SPLINE
SPL {X  -145.877, Y  +737.201, Z    +0.000, E1   -34.468, E3 +267717.611}
SPL {X  -152.550, Y  +719.721, Z    +0.000, E1   -27.728, E3 +267733.100}
SPL {X  -157.145, Y  +701.536, Z    +0.000, E1   -19.368, E3 +267742.554}
SPL {X  -159.035, Y  +688.952, Z    +0.000, E1   -12.676, E3 +267746.596}
SPL {X  -159.756, Y  +680.154, Z    +0.000, E1    -7.520, E3 +267748.322}
SPL {X  -159.986, Y  +672.560, Z    +0.000, E1    -2.636, E3 +267749.220}
SPL {X  -159.990, Y  +668.344, Z    +0.000, E1    +0.618, E3 +267749.486}
SPL {X  -159.990, Y  +664.070, Z    +0.000, E1    +5.025, E3 +267749.815}
SPL {X  -159.990, Y  +656.953, Z    +0.000, E1   +13.960, E3 +267750.881}
SPL {X  -159.990, Y  +644.589, Z    +0.000, E1   +29.011, E3 +267754.293}
SPL {X  -159.990, Y  +605.095, Z    +0.000, E1   +49.514, E3 +267779.383}
SPL {X  -159.990, Y  +543.998, Z    +0.000, E1   +54.483, E3 +267845.373}
SPL {X  -159.990, Y  +535.878, Z    +0.000, E1   +54.465, E3 +267857.708}
SPL {X  -159.990, Y  +529.394, Z    +0.000, E1   +54.464, E3 +267867.538}
SPL {X  -159.990, Y  +521.536, Z    +0.000, E1   +54.480, E3 +267879.419}
SPL {X  -159.990, Y  +514.089, Z    +0.000, E1   +54.461, E3 +267890.732}
SPL {X  -159.990, Y  +506.373, Z    +0.000, E1   +54.484, E3 +267902.368}
SPL {X  -159.990, Y  +497.571, Z    +0.000, E1   +54.478, E3 +267915.711}
SPL {X  -159.990, Y  +490.343, Z    +0.000, E1   +54.468, E3 +267926.676}
SPL {X  -159.990, Y  +483.191, Z    +0.000, E1   +54.478, E3 +267937.492}
SPL {X  -159.990, Y  +471.543, Z    +0.000, E1   +55.096, E3 +267951.120}
SPL {X  -159.990, Y  +443.253, Z    +0.000, E1   +59.297, E3 +267962.552}
SPL {X  -159.990, Y  +438.044, Z    +0.000, E1   +58.687, E3 +267973.407}
SPL {X  -159.990, Y  +431.936, Z    +0.000, E1   +57.955, E3 +267986.227}
SPL {X  -159.990, Y  +427.860, Z    +0.000, E1   +57.091, E3 +267997.291}
SPL {X  -159.990, Y  +424.653, Z    +0.000, E1   +55.901, E3 +268009.596}
SPL {X  -159.990, Y  +418.232, Z    +0.000, E1   +55.048, E3 +268024.389}
SPL {X  -159.990, Y  +410.722, Z    +0.000, E1   +54.900, E3 +268036.372}
SPL {X  -159.990, Y  +402.790, Z    +0.000, E1   +54.930, E3 +268048.147}
SPL {X  -159.990, Y  +391.119, Z    +0.000, E1   +54.948, E3 +268065.524}
SPL {X  -159.951, Y  +378.972, Z    +0.000, E1   +54.929, E3 +268083.703}
SPL {X  -159.499, Y  +369.977, Z    +0.000, E1   +54.827, E3 +268097.615}
SPL {X  -158.803, Y  +363.045, Z    +0.000, E1   +54.709, E3 +268108.684}
SPL {X  -157.966, Y  +357.131, Z    +0.000, E1   +54.559, E3 +268118.386}
SPL {X  -156.775, Y  +350.586, Z    +0.000, E1   +54.373, E3 +268129.360}
SPL {X  -155.027, Y  +342.959, Z    +0.000, E1   +54.074, E3 +268142.533}
SPL {X  -152.882, Y  +335.340, Z    +0.000, E1   +53.695, E3 +268156.076}
SPL {X  -151.019, Y  +329.680, Z    +0.000, E1   +53.334, E3 +268166.433}
SPL {X  -149.351, Y  +325.131, Z    +0.000, E1   +53.025, E3 +268174.877}
SPL {X  -147.860, Y  +321.391, Z    +0.000, E1   +52.740, E3 +268181.930}
SPL {X  -145.914, Y  +316.881, Z    +0.000, E1   +52.402, E3 +268190.499}
SPL {X  -142.795, Y  +310.344, Z    +0.000, E1   +51.829, E3 +268203.155}
SPL {X  -132.354, Y  +292.616, Z    +0.000, E1   +44.164, E3 +268301.567}
ENDSPLINE

SPLINE
SPL {X  -150.910, Y  +329.369, Z    +0.000, E1   +29.678, E3 +268373.963}
SPL {X  -156.396, Y  +348.778, Z    +0.000, E1   +21.134, E3 +268385.606}
SPL {X  -158.554, Y  +361.116, Z    +0.000, E1   +14.883, E3 +268390.060}
SPL {X  -159.881, Y  +376.607, Z    +0.000, E1    +5.865, E3 +268393.469}
SPL {X  -159.990, Y  +383.659, Z    +0.000, E1    +1.050, E3 +268394.150}
SPL {X  -159.990, Y  +387.327, Z    +0.000, E1    -2.137, E3 +268394.383}
SPL {X  -159.990, Y  +390.622, Z    +0.000, E1    -5.876, E3 +268394.676}
SPL {X  -159.990, Y  +394.493, Z    +0.000, E1   -10.512, E3 +268395.199}
SPL {X  -159.990, Y  +401.377, Z    +0.000, E1   -19.398, E3 +268396.653}
SPL {X  -159.990, Y  +411.365, Z    +0.000, E1   -30.630, E3 +268399.862}
SPL {X  -159.990, Y  +450.467, Z    +0.000, E1   -50.183, E3 +268423.511}
SPL {X  -159.990, Y  +509.934, Z    +0.000, E1   -54.923, E3 +268486.130}
SPL {X  -159.990, Y  +516.848, Z    +0.000, E1   -54.930, E3 +268496.418}
SPL {X  -159.990, Y  +524.818, Z    +0.000, E1   -54.933, E3 +268508.290}
SPL {X  -159.990, Y  +532.100, Z    +0.000, E1   -54.924, E3 +268519.143}
SPL {X  -159.990, Y  +539.391, Z    +0.000, E1   -54.933, E3 +268529.995}
SPL {X  -159.990, Y  +546.283, Z    +0.000, E1   -54.924, E3 +268540.266}
SPL {X  -159.990, Y  +553.734, Z    +0.000, E1   -54.938, E3 +268551.353}
SPL {X  -159.990, Y  +564.956, Z    +0.000, E1   -54.973, E3 +268568.024}
SPL {X  -159.990, Y  +577.902, Z    +0.000, E1   -54.969, E3 +268587.314}
SPL {X  -159.990, Y  +588.063, Z    +0.000, E1   -54.931, E3 +268602.505}
SPL {X  -159.990, Y  +595.273, Z    +0.000, E1   -54.928, E3 +268613.228}
SPL {X  -159.990, Y  +602.326, Z    +0.000, E1   -54.932, E3 +268623.729}
SPL {X  -159.990, Y  +610.296, Z    +0.000, E1   -54.937, E3 +268635.598}
SPL {X  -159.990, Y  +618.534, Z    +0.000, E1   -54.942, E3 +268647.835}
SPL {X  -159.990, Y  +628.178, Z    +0.000, E1   -54.959, E3 +268662.166}
SPL {X  -159.990, Y  +638.304, Z    +0.000, E1   -54.952, E3 +268677.255}
SPL {X  -159.990, Y  +648.272, Z    +0.000, E1   -54.961, E3 +268692.064}
SPL {X  -159.990, Y  +655.990, Z    +0.000, E1   -54.930, E3 +268703.612}
SPL {X  -159.990, Y  +665.734, Z    +0.000, E1   -54.984, E3 +268718.063}
SPL {X  -159.827, Y  +678.718, Z    +0.000, E1   -54.950, E3 +268737.591}
SPL {X  -159.222, Y  +687.156, Z    +0.000, E1   -54.792, E3 +268750.902}
SPL {X  -158.388, Y  +694.082, Z    +0.000, E1   -54.679, E3 +268762.040}
SPL {X  -157.277, Y  +700.838, Z    +0.000, E1   -54.465, E3 +268773.297}
SPL {X  -156.153, Y  +706.327, Z    +0.000, E1   -54.274, E3 +268782.633}
SPL {X  -154.917, Y  +711.470, Z    +0.000, E1   -54.052, E3 +268791.584}
SPL {X  -153.204, Y  +717.603, Z    +0.000, E1   -53.775, E3 +268802.430}
SPL {X  -151.355, Y  +723.351, Z    +0.000, E1   -53.415, E3 +268812.901}
SPL {X  -149.371, Y  +728.816, Z    +0.000, E1   -53.074, E3 +268822.992}
SPL {X  -147.376, Y  +733.767, Z    +0.000, E1   -52.671, E3 +268832.394}
SPL {X  -145.158, Y  +738.775, Z    +0.000, E1   -52.288, E3 +268841.945}
SPL {X  -142.385, Y  +744.461, Z    +0.000, E1   -51.729, E3 +268853.057}
SPL {X  -132.301, Y  +761.463, Z    +0.000, E1   -45.510, E3 +268930.796}
ENDSPLINE

SPLINE
SPL {X  -145.877, Y  +737.201, Z    +0.000, E1   -34.468, E3 +269013.907}
SPL {X  -152.550, Y  +719.721, Z    +0.000, E1   -27.728, E3 +269029.396}
SPL {X  -157.145, Y  +701.536, Z    +0.000, E1   -19.368, E3 +269038.851}
SPL {X  -159.035, Y  +688.952, Z    +0.000, E1   -12.676, E3 +269042.892}
SPL {X  -159.756, Y  +680.154, Z    +0.000, E1    -7.520, E3 +269044.618}
SPL {X  -159.986, Y  +672.560, Z    +0.000, E1    -2.636, E3 +269045.516}
SPL {X  -159.990, Y  +668.344, Z    +0.000, E1    +0.618, E3 +269045.782}
SPL {X  -159.990, Y  +664.070, Z    +0.000, E1    +5.025, E3 +269046.111}
SPL {X  -159.990, Y  +656.953, Z    +0.000, E1   +13.960, E3 +269047.177}
SPL {X  -159.990, Y  +644.589, Z    +0.000, E1   +29.011, E3 +269050.589}
SPL {X  -159.990, Y  +605.095, Z    +0.000, E1   +49.514, E3 +269075.680}
SPL {X  -159.990, Y  +546.155, Z    +0.000, E1   +54.461, E3 +269138.438}
SPL {X  -159.990, Y  +537.700, Z    +0.000, E1   +54.492, E3 +269151.202}
SPL {X  -159.990, Y  +529.394, Z    +0.000, E1   +54.464, E3 +269163.834}
SPL {X  -159.990, Y  +521.536, Z    +0.000, E1   +54.480, E3 +269175.715}
SPL {X  -159.990, Y  +514.089, Z    +0.000, E1   +54.461, E3 +269187.028}
SPL {X  -159.990, Y  +506.373, Z    +0.000, E1   +54.484, E3 +269198.664}
SPL {X  -159.990, Y  +497.571, Z    +0.000, E1   +54.478, E3 +269212.007}
SPL {X  -159.990, Y  +490.343, Z    +0.000, E1   +54.468, E3 +269222.972}
SPL {X  -159.990, Y  +483.191, Z    +0.000, E1   +54.478, E3 +269233.789}
SPL {X  -159.990, Y  +475.502, Z    +0.000, E1   +54.476, E3 +269245.438}
SPL {X  -159.990, Y  +448.520, Z    +0.000, E1   +58.543, E3 +269257.067}
SPL {X  -159.990, Y  +438.044, Z    +0.000, E1   +58.687, E3 +269269.704}
SPL {X  -159.990, Y  +431.936, Z    +0.000, E1   +57.955, E3 +269282.523}
SPL {X  -159.990, Y  +427.860, Z    +0.000, E1   +57.091, E3 +269293.587}
SPL {X  -159.990, Y  +424.653, Z    +0.000, E1   +55.901, E3 +269305.892}
SPL {X  -159.990, Y  +418.232, Z    +0.000, E1   +55.048, E3 +269320.685}
SPL {X  -159.990, Y  +410.722, Z    +0.000, E1   +54.900, E3 +269332.668}
SPL {X  -159.990, Y  +402.790, Z    +0.000, E1   +54.930, E3 +269344.443}
SPL {X  -159.990, Y  +392.953, Z    +0.000, E1   +54.918, E3 +269359.137}
SPL {X  -159.990, Y  +383.354, Z    +0.000, E1   +54.920, E3 +269373.447}
SPL {X  -159.860, Y  +376.053, Z    +0.000, E1   +54.872, E3 +269384.507}
SPL {X  -159.499, Y  +369.977, Z    +0.000, E1   +54.827, E3 +269393.911}
SPL {X  -158.803, Y  +363.045, Z    +0.000, E1   +54.709, E3 +269404.980}
SPL {X  -157.732, Y  +355.717, Z    +0.000, E1   +54.540, E3 +269417.002}
SPL {X  -156.235, Y  +348.039, Z    +0.000, E1   +54.281, E3 +269430.014}
SPL {X  -154.716, Y  +341.761, Z    +0.000, E1   +53.995, E3 +269440.971}
SPL {X  -152.882, Y  +335.340, Z    +0.000, E1   +53.695, E3 +269452.372}
SPL {X  -151.019, Y  +329.680, Z    +0.000, E1   +53.334, E3 +269462.729}
SPL {X  -149.351, Y  +325.131, Z    +0.000, E1   +53.025, E3 +269471.173}
SPL {X  -147.860, Y  +321.391, Z    +0.000, E1   +52.740, E3 +269478.226}
SPL {X  -145.914, Y  +316.881, Z    +0.000, E1   +52.402, E3 +269486.796}
SPL {X  -142.795, Y  +310.344, Z    +0.000, E1   +51.829, E3 +269499.451}
SPL {X  -132.354, Y  +292.616, Z    +0.000, E1   +44.164, E3 +269597.864}
ENDSPLINE

SPLINE
SPL {X  -150.910, Y  +329.369, Z    +0.000, E1   +29.678, E3 +269670.259}
SPL {X  -156.829, Y  +350.854, Z    +0.000, E1   +20.141, E3 +269682.812}
SPL {X  -159.049, Y  +365.169, Z    +0.000, E1   +12.580, E3 +269687.556}
SPL {X  -159.776, Y  +374.231, Z    +0.000, E1    +7.281, E3 +269689.442}
SPL {X  -159.986, Y  +381.380, Z    +0.000, E1    +2.685, E3 +269690.288}
SPL {X  -159.990, Y  +384.493, Z    +0.000, E1    +0.324, E3 +269690.496}
SPL {X  -159.990, Y  +387.327, Z    +0.000, E1    -2.137, E3 +269690.679}
SPL {X  -159.990, Y  +392.053, Z    +0.000, E1    -7.477, E3 +269691.144}
SPL {X  -159.990, Y  +396.158, Z    +0.000, E1   -12.775, E3 +269691.769}
SPL {X  -159.990, Y  +401.377, Z    +0.000, E1   -19.398, E3 +269692.950}
SPL {X  -159.990, Y  +411.365, Z    +0.000, E1   -30.630, E3 +269696.158}
SPL {X  -159.990, Y  +450.467, Z    +0.000, E1   -50.183, E3 +269719.807}
SPL {X  -159.990, Y  +509.934, Z    +0.000, E1   -54.923, E3 +269782.426}
SPL {X  -159.990, Y  +516.848, Z    +0.000, E1   -54.930, E3 +269792.714}
SPL {X  -159.990, Y  +524.818, Z    +0.000, E1   -54.933, E3 +269804.586}
SPL {X  -159.990, Y  +532.100, Z    +0.000, E1   -54.924, E3 +269815.439}
SPL {X  -159.990, Y  +539.391, Z    +0.000, E1   -54.933, E3 +269826.291}
SPL {X  -159.990, Y  +546.283, Z    +0.000, E1   -54.924, E3 +269836.562}
SPL {X  -159.990, Y  +553.734, Z    +0.000, E1   -54.938, E3 +269847.649}
SPL {X  -159.990, Y  +560.983, Z    +0.000, E1   -54.918, E3 +269858.487}
SPL {X  -159.990, Y  +567.462, Z    +0.000, E1   -54.929, E3 +269868.122}
SPL {X  -159.990, Y  +575.140, Z    +0.000, E1   -54.928, E3 +269879.554}
SPL {X  -159.990, Y  +581.046, Z    +0.000, E1   -54.920, E3 +269888.366}
SPL {X  -159.990, Y  +588.063, Z    +0.000, E1   -54.931, E3 +269898.801}
SPL {X  -159.990, Y  +595.273, Z    +0.000, E1   -54.928, E3 +269909.525}
SPL {X  -159.990, Y  +602.326, Z    +0.000, E1   -54.932, E3 +269920.025}
SPL {X  -159.990, Y  +610.296, Z    +0.000, E1   -54.937, E3 +269931.894}
SPL {X  -159.990, Y  +618.534, Z    +0.000, E1   -54.942, E3 +269944.131}
SPL {X  -159.990, Y  +625.928, Z    +0.000, E1   -54.931, E3 +269955.157}
SPL {X  -159.990, Y  +633.423, Z    +0.000, E1   -54.943, E3 +269966.299}
SPL {X  -159.990, Y  +643.352, Z    +0.000, E1   -54.966, E3 +269981.034}
SPL {X  -159.990, Y  +650.756, Z    +0.000, E1   -54.931, E3 +269992.101}
SPL {X  -159.990, Y  +658.525, Z    +0.000, E1   -54.959, E3 +270003.637}
SPL {X  -159.990, Y  +667.903, Z    +0.000, E1   -54.941, E3 +270017.668}
SPL {X  -159.953, Y  +674.920, Z    +0.000, E1   -54.918, E3 +270028.171}
SPL {X  -159.714, Y  +680.893, Z    +0.000, E1   -54.890, E3 +270037.311}
SPL {X  -159.222, Y  +687.156, Z    +0.000, E1   -54.792, E3 +270047.198}
SPL {X  -158.388, Y  +694.082, Z    +0.000, E1   -54.679, E3 +270058.336}
SPL {X  -157.277, Y  +700.838, Z    +0.000, E1   -54.465, E3 +270069.593}
SPL {X  -156.153, Y  +706.327, Z    +0.000, E1   -54.274, E3 +270078.929}
SPL {X  -154.917, Y  +711.470, Z    +0.000, E1   -54.052, E3 +270087.880}
SPL {X  -153.204, Y  +717.603, Z    +0.000, E1   -53.775, E3 +270098.726}
SPL {X  -151.355, Y  +723.351, Z    +0.000, E1   -53.415, E3 +270109.198}
SPL {X  -149.371, Y  +728.816, Z    +0.000, E1   -53.074, E3 +270119.288}
SPL {X  -146.631, Y  +735.501, Z    +0.000, E1   -52.568, E3 +270131.949}
SPL {X  -144.428, Y  +740.329, Z    +0.000, E1   -52.109, E3 +270141.303}
SPL {X  -142.385, Y  +744.461, Z    +0.000, E1   -51.729, E3 +270149.354}
SPL {X  -132.301, Y  +761.463, Z    +0.000, E1   -45.510, E3 +270227.092}
ENDSPLINE

SPLINE
SPL {X  -145.877, Y  +737.201, Z    +0.000, E1   -34.468, E3 +270310.203}
SPL {X  -152.550, Y  +719.721, Z    +0.000, E1   -27.728, E3 +270325.692}
SPL {X  -157.145, Y  +701.536, Z    +0.000, E1   -19.368, E3 +270335.147}
SPL {X  -159.035, Y  +688.952, Z    +0.000, E1   -12.676, E3 +270339.188}
SPL {X  -159.756, Y  +680.154, Z    +0.000, E1    -7.520, E3 +270340.914}
SPL {X  -159.986, Y  +672.560, Z    +0.000, E1    -2.636, E3 +270341.813}
SPL {X  -159.990, Y  +668.344, Z    +0.000, E1    +0.618, E3 +270342.079}
SPL {X  -159.990, Y  +664.070, Z    +0.000, E1    +5.025, E3 +270342.407}
SPL {X  -159.990, Y  +656.953, Z    +0.000, E1   +13.960, E3 +270343.474}
SPL {X  -159.990, Y  +644.589, Z    +0.000, E1   +29.011, E3 +270346.885}
SPL {X  -159.990, Y  +605.095, Z    +0.000, E1   +49.514, E3 +270371.976}
SPL {X  -159.990, Y  +543.998, Z    +0.000, E1   +54.483, E3 +270437.966}
SPL {X  -159.990, Y  +535.878, Z    +0.000, E1   +54.465, E3 +270450.301}
SPL {X  -159.990, Y  +529.394, Z    +0.000, E1   +54.464, E3 +270460.130}
SPL {X  -159.990, Y  +521.536, Z    +0.000, E1   +54.480, E3 +270472.012}
SPL {X  -159.990, Y  +514.089, Z    +0.000, E1   +54.461, E3 +270483.324}
SPL {X  -159.990, Y  +506.373, Z    +0.000, E1   +54.484, E3 +270494.961}
SPL {X  -159.990, Y  +497.571, Z    +0.000, E1   +54.478, E3 +270508.304}
SPL {X  -159.990, Y  +490.343, Z    +0.000, E1   +54.468, E3 +270519.269}
SPL {X  -159.990, Y  +483.191, Z    +0.000, E1   +54.478, E3 +270530.085}
SPL {X  -159.990, Y  +471.543, Z    +0.000, E1   +55.096, E3 +270543.713}
SPL {X  -159.990, Y  +443.253, Z    +0.000, E1   +59.297, E3 +270555.145}
SPL {X  -159.990, Y  +438.044, Z    +0.000, E1   +58.687, E3 +270566.000}
SPL {X  -159.990, Y  +431.936, Z    +0.000, E1   +57.955, E3 +270578.819}
SPL {X  -159.990, Y  +427.293, Z    +0.000, E1   +56.830, E3 +270592.525}
SPL {X  -159.990, Y  +423.841, Z    +0.000, E1   +55.679, E3 +270604.627}
SPL {X  -159.990, Y  +419.589, Z    +0.000, E1   +55.096, E3 +270614.552}
SPL {X  -159.990, Y  +412.636, Z    +0.000, E1   +54.925, E3 +270626.064}
SPL {X  -159.990, Y  +405.235, Z    +0.000, E1   +54.902, E3 +270637.134}
SPL {X  -159.990, Y  +400.284, Z    +0.000, E1   +54.897, E3 +270644.528}
SPL {X  -159.990, Y  +392.953, Z    +0.000, E1   +54.918, E3 +270655.433}
SPL {X  -159.990, Y  +383.354, Z    +0.000, E1   +54.920, E3 +270669.743}
SPL {X  -159.860, Y  +376.053, Z    +0.000, E1   +54.872, E3 +270680.803}
SPL {X  -159.499, Y  +369.977, Z    +0.000, E1   +54.827, E3 +270690.208}
SPL {X  -158.803, Y  +363.045, Z    +0.000, E1   +54.709, E3 +270701.276}
SPL {X  -157.966, Y  +357.131, Z    +0.000, E1   +54.559, E3 +270710.979}
SPL {X  -156.775, Y  +350.586, Z    +0.000, E1   +54.373, E3 +270721.953}
SPL {X  -155.027, Y  +342.959, Z    +0.000, E1   +54.074, E3 +270735.126}
SPL {X  -153.580, Y  +337.668, Z    +0.000, E1   +53.781, E3 +270744.549}
SPL {X  -151.643, Y  +331.497, Z    +0.000, E1   +53.493, E3 +270755.628}
SPL {X  -148.682, Y  +323.421, Z    +0.000, E1   +52.939, E3 +270770.628}
SPL {X  -145.914, Y  +316.881, Z    +0.000, E1   +52.402, E3 +270783.092}
SPL {X  -143.679, Y  +312.121, Z    +0.000, E1   +51.954, E3 +270792.337}
SPL {X  -141.812, Y  +308.430, Z    +0.000, E1   +51.590, E3 +270799.569}
SPL {X  -132.354, Y  +292.616, Z    +0.000, E1   +44.164, E3 +270894.160}
ENDSPLINE

SPLINE
SPL {X  -150.910, Y  +329.369, Z    +0.000, E1   +29.678, E3 +270966.555}
SPL {X  -156.829, Y  +350.854, Z    +0.000, E1   +20.141, E3 +270979.108}
SPL {X  -159.049, Y  +365.169, Z    +0.000, E1   +12.580, E3 +270983.852}
SPL {X  -159.881, Y  +376.607, Z    +0.000, E1    +5.865, E3 +270986.062}
SPL {X  -159.990, Y  +382.403, Z    +0.000, E1    +1.910, E3 +270986.667}
SPL {X  -159.990, Y  +385.261, Z    +0.000, E1    -0.259, E3 +270986.838}
SPL {X  -159.990, Y  +389.002, Z    +0.000, E1    -3.890, E3 +270987.116}
SPL {X  -159.990, Y  +394.493, Z    +0.000, E1   -10.512, E3 +270987.792}
SPL {X  -159.990, Y  +401.377, Z    +0.000, E1   -19.398, E3 +270989.246}
SPL {X  -159.990, Y  +411.365, Z    +0.000, E1   -30.630, E3 +270992.454}
SPL {X  -159.990, Y  +450.467, Z    +0.000, E1   -50.183, E3 +271016.103}
SPL {X  -159.990, Y  +509.934, Z    +0.000, E1   -54.923, E3 +271078.722}
SPL {X  -159.990, Y  +516.848, Z    +0.000, E1   -54.930, E3 +271089.010}
SPL {X  -159.990, Y  +524.818, Z    +0.000, E1   -54.933, E3 +271100.882}
SPL {X  -159.990, Y  +532.100, Z    +0.000, E1   -54.924, E3 +271111.735}
SPL {X  -159.990, Y  +539.391, Z    +0.000, E1   -54.933, E3 +271122.587}
SPL {X  -159.990, Y  +546.283, Z    +0.000, E1   -54.924, E3 +271132.859}
SPL {X  -159.990, Y  +553.734, Z    +0.000, E1   -54.938, E3 +271143.946}
SPL {X  -159.990, Y  +564.956, Z    +0.000, E1   -54.973, E3 +271160.617}
SPL {X  -159.990, Y  +577.902, Z    +0.000, E1   -54.969, E3 +271179.907}
SPL {X  -159.990, Y  +588.063, Z    +0.000, E1   -54.931, E3 +271195.097}
SPL {X  -159.990, Y  +595.273, Z    +0.000, E1   -54.928, E3 +271205.821}
SPL {X  -159.990, Y  +602.326, Z    +0.000, E1   -54.932, E3 +271216.321}
SPL {X  -159.990, Y  +610.296, Z    +0.000, E1   -54.937, E3 +271228.191}
SPL {X  -159.990, Y  +618.534, Z    +0.000, E1   -54.942, E3 +271240.428}
SPL {X  -159.990, Y  +625.928, Z    +0.000, E1   -54.931, E3 +271251.453}
SPL {X  -159.990, Y  +633.423, Z    +0.000, E1   -54.943, E3 +271262.595}
SPL {X  -159.990, Y  +640.333, Z    +0.000, E1   -54.927, E3 +271272.909}
SPL {X  -159.990, Y  +648.272, Z    +0.000, E1   -54.961, E3 +271284.657}
SPL {X  -159.990, Y  +655.990, Z    +0.000, E1   -54.930, E3 +271296.204}
SPL {X  -159.990, Y  +665.734, Z    +0.000, E1   -54.984, E3 +271310.655}
SPL {X  -159.827, Y  +678.718, Z    +0.000, E1   -54.950, E3 +271330.184}
SPL {X  -159.222, Y  +687.156, Z    +0.000, E1   -54.792, E3 +271343.494}
SPL {X  -158.388, Y  +694.082, Z    +0.000, E1   -54.679, E3 +271354.632}
SPL {X  -157.277, Y  +700.838, Z    +0.000, E1   -54.465, E3 +271365.889}
SPL {X  -156.153, Y  +706.327, Z    +0.000, E1   -54.274, E3 +271375.225}
SPL {X  -154.917, Y  +711.470, Z    +0.000, E1   -54.052, E3 +271384.177}
SPL {X  -153.204, Y  +717.603, Z    +0.000, E1   -53.775, E3 +271395.023}
SPL {X  -150.773, Y  +725.019, Z    +0.000, E1   -53.343, E3 +271408.516}
SPL {X  -148.029, Y  +732.198, Z    +0.000, E1   -52.831, E3 +271421.953}
SPL {X  -145.158, Y  +738.775, Z    +0.000, E1   -52.288, E3 +271434.538}
SPL {X  -142.385, Y  +744.461, Z    +0.000, E1   -51.729, E3 +271445.650}
SPL {X  -132.301, Y  +761.463, Z    +0.000, E1   -45.510, E3 +271523.389}
ENDSPLINE

SPLINE
SPL {X  -145.877, Y  +737.201, Z    +0.000, E1   -34.468, E3 +271606.500}
SPL {X  -152.550, Y  +719.721, Z    +0.000, E1   -27.728, E3 +271621.989}
SPL {X  -157.145, Y  +701.536, Z    +0.000, E1   -19.368, E3 +271631.443}
SPL {X  -159.035, Y  +688.952, Z    +0.000, E1   -12.676, E3 +271635.484}
SPL {X  -159.873, Y  +677.622, Z    +0.000, E1    -6.008, E3 +271637.556}
SPL {X  -159.990, Y  +670.381, Z    +0.000, E1    -1.064, E3 +271638.257}
SPL {X  -159.990, Y  +666.603, Z    +0.000, E1    +2.256, E3 +271638.488}
SPL {X  -159.990, Y  +661.750, Z    +0.000, E1    +7.880, E3 +271638.961}
SPL {X  -159.990, Y  +657.656, Z    +0.000, E1   +13.276, E3 +271639.606}
SPL {X  -159.990, Y  +652.023, Z    +0.000, E1   +20.449, E3 +271640.894}
SPL {X  -159.990, Y  +641.935, Z    +0.000, E1   +31.848, E3 +271644.066}
SPL {X  -159.990, Y  +605.095, Z    +0.000, E1   +49.514, E3 +271668.272}
SPL {X  -159.990, Y  +543.998, Z    +0.000, E1   +54.483, E3 +271734.262}
SPL {X  -159.990, Y  +535.878, Z    +0.000, E1   +54.465, E3 +271746.597}
SPL {X  -159.990, Y  +529.394, Z    +0.000, E1   +54.464, E3 +271756.426}
SPL {X  -159.990, Y  +521.536, Z    +0.000, E1   +54.480, E3 +271768.308}
SPL {X  -159.990, Y  +512.119, Z    +0.000, E1   +54.487, E3 +271782.554}
SPL {X  -159.990, Y  +504.581, Z    +0.000, E1   +54.460, E3 +271794.013}
SPL {X  -159.990, Y  +497.571, Z    +0.000, E1   +54.478, E3 +271804.600}
SPL {X  -159.990, Y  +490.343, Z    +0.000, E1   +54.468, E3 +271815.565}
SPL {X  -159.990, Y  +483.191, Z    +0.000, E1   +54.478, E3 +271826.381}
SPL {X  -159.990, Y  +471.543, Z    +0.000, E1   +55.096, E3 +271840.009}
SPL {X  -159.990, Y  +443.253, Z    +0.000, E1   +59.297, E3 +271851.441}
SPL {X  -159.990, Y  +438.044, Z    +0.000, E1   +58.687, E3 +271862.296}
SPL {X  -159.990, Y  +431.936, Z    +0.000, E1   +57.955, E3 +271875.116}
SPL {X  -159.990, Y  +427.293, Z    +0.000, E1   +56.830, E3 +271888.822}
SPL {X  -159.990, Y  +423.841, Z    +0.000, E1   +55.679, E3 +271900.924}
SPL {X  -159.990, Y  +418.232, Z    +0.000, E1   +55.048, E3 +271913.278}
SPL {X  -159.990, Y  +410.722, Z    +0.000, E1   +54.900, E3 +271925.261}
SPL {X  -159.990, Y  +402.790, Z    +0.000, E1   +54.930, E3 +271937.036}
SPL {X  -159.990, Y  +392.953, Z    +0.000, E1   +54.918, E3 +271951.729}
SPL {X  -159.990, Y  +383.354, Z    +0.000, E1   +54.920, E3 +271966.039}
SPL {X  -159.769, Y  +374.091, Z    +0.000, E1   +54.882, E3 +271980.072}
SPL {X  -158.996, Y  +364.689, Z    +0.000, E1   +54.773, E3 +271994.868}
SPL {X  -157.732, Y  +355.717, Z    +0.000, E1   +54.540, E3 +272009.595}
SPL {X  -156.235, Y  +348.039, Z    +0.000, E1   +54.281, E3 +272022.606}
SPL {X  -154.716, Y  +341.761, Z    +0.000, E1   +53.995, E3 +272033.563}
SPL {X  -152.882, Y  +335.340, Z    +0.000, E1   +53.695, E3 +272044.965}
SPL {X  -151.019, Y  +329.680, Z    +0.000, E1   +53.334, E3 +272055.322}
SPL {X  -148.682, Y  +323.421, Z    +0.000, E1   +52.939, E3 +272066.924}
SPL {X  -145.914, Y  +316.881, Z    +0.000, E1   +52.402, E3 +272079.388}
SPL {X  -142.795, Y  +310.344, Z    +0.000, E1   +51.829, E3 +272092.044}
SPL {X  -132.354, Y  +292.616, Z    +0.000, E1   +44.164, E3 +272190.456}
ENDSPLINE

SPLINE
SPL {X  -150.910, Y  +329.369, Z    +0.000, E1   +29.678, E3 +272262.852}
SPL {X  -156.829, Y  +350.854, Z    +0.000, E1   +20.141, E3 +272275.405}
SPL {X  -159.049, Y  +365.169, Z    +0.000, E1   +12.580, E3 +272280.149}
SPL {X  -159.776, Y  +374.231, Z    +0.000, E1    +7.281, E3 +272282.035}
SPL {X  -159.986, Y  +381.380, Z    +0.000, E1    +2.685, E3 +272282.881}
SPL {X  -159.990, Y  +385.261, Z    +0.000, E1    -0.259, E3 +272283.134}
SPL {X  -159.990, Y  +388.094, Z    +0.000, E1    -3.012, E3 +272283.326}
SPL {X  -159.990, Y  +392.053, Z    +0.000, E1    -7.477, E3 +272283.736}
SPL {X  -159.990, Y  +396.158, Z    +0.000, E1   -12.775, E3 +272284.362}
SPL {X  -159.990, Y  +401.377, Z    +0.000, E1   -19.398, E3 +272285.542}
SPL {X  -159.990, Y  +411.365, Z    +0.000, E1   -30.630, E3 +272288.751}
SPL {X  -159.990, Y  +450.467, Z    +0.000, E1   -50.183, E3 +272312.400}
SPL {X  -159.990, Y  +509.934, Z    +0.000, E1   -54.923, E3 +272375.018}
SPL {X  -159.990, Y  +516.848, Z    +0.000, E1   -54.930, E3 +272385.307}
SPL {X  -159.990, Y  +524.818, Z    +0.000, E1   -54.933, E3 +272397.178}
SPL {X  -159.990, Y  +532.100, Z    +0.000, E1   -54.924, E3 +272408.031}
SPL {X  -159.990, Y  +539.391, Z    +0.000, E1   -54.933, E3 +272418.883}
SPL {X  -159.990, Y  +546.283, Z    +0.000, E1   -54.924, E3 +272429.155}
SPL {X  -159.990, Y  +553.734, Z    +0.000, E1   -54.938, E3 +272440.242}
SPL {X  -159.990, Y  +564.956, Z    +0.000, E1   -54.973, E3 +272456.913}
SPL {X  -159.990, Y  +575.140, Z    +0.000, E1   -54.928, E3 +272472.146}
SPL {X  -159.990, Y  +581.046, Z    +0.000, E1   -54.920, E3 +272480.959}
SPL {X  -159.990, Y  +588.063, Z    +0.000, E1   -54.931, E3 +272491.394}
SPL {X  -159.990, Y  +595.273, Z    +0.000, E1   -54.928, E3 +272502.117}
SPL {X  -159.990, Y  +602.326, Z    +0.000, E1   -54.932, E3 +272512.618}
SPL {X  -159.990, Y  +610.296, Z    +0.000, E1   -54.937, E3 +272524.487}
SPL {X  -159.990, Y  +618.534, Z    +0.000, E1   -54.942, E3 +272536.724}
SPL {X  -159.990, Y  +625.928, Z    +0.000, E1   -54.931, E3 +272547.749}
SPL {X  -159.990, Y  +633.423, Z    +0.000, E1   -54.943, E3 +272558.891}
SPL {X  -159.990, Y  +640.333, Z    +0.000, E1   -54.927, E3 +272569.206}
SPL {X  -159.990, Y  +648.272, Z    +0.000, E1   -54.961, E3 +272580.953}
SPL {X  -159.990, Y  +658.525, Z    +0.000, E1   -54.959, E3 +272596.229}
SPL {X  -159.990, Y  +667.903, Z    +0.000, E1   -54.941, E3 +272610.261}
SPL {X  -159.827, Y  +678.718, Z    +0.000, E1   -54.950, E3 +272626.480}
SPL {X  -159.222, Y  +687.156, Z    +0.000, E1   -54.792, E3 +272639.791}
SPL {X  -158.388, Y  +694.082, Z    +0.000, E1   -54.679, E3 +272650.928}
SPL {X  -157.277, Y  +700.838, Z    +0.000, E1   -54.465, E3 +272662.186}
SPL {X  -156.153, Y  +706.327, Z    +0.000, E1   -54.274, E3 +272671.522}
SPL {X  -154.917, Y  +711.470, Z    +0.000, E1   -54.052, E3 +272680.473}
SPL {X  -153.204, Y  +717.603, Z    +0.000, E1   -53.775, E3 +272691.319}
SPL {X  -150.773, Y  +725.019, Z    +0.000, E1   -53.343, E3 +272704.812}
SPL {X  -148.029, Y  +732.198, Z    +0.000, E1   -52.831, E3 +272718.249}
SPL {X  -145.158, Y  +738.775, Z    +0.000, E1   -52.288, E3 +272730.834}
SPL {X  -142.385, Y  +744.461, Z    +0.000, E1   -51.729, E3 +272741.946}
SPL {X  -132.301, Y  +761.463, Z    +0.000, E1   -45.510, E3 +272819.685}
ENDSPLINE

SPLINE
SPL {X  -145.877, Y  +737.201, Z    +0.000, E1   -34.468, E3 +272902.796}
SPL {X  -152.550, Y  +719.721, Z    +0.000, E1   -27.728, E3 +272918.285}
SPL {X  -157.145, Y  +701.536, Z    +0.000, E1   -19.368, E3 +272927.740}
SPL {X  -159.035, Y  +688.952, Z    +0.000, E1   -12.676, E3 +272931.781}
SPL {X  -159.756, Y  +680.154, Z    +0.000, E1    -7.520, E3 +272933.507}
SPL {X  -159.986, Y  +672.560, Z    +0.000, E1    -2.636, E3 +272934.405}
SPL {X  -159.990, Y  +668.344, Z    +0.000, E1    +0.618, E3 +272934.671}
SPL {X  -159.990, Y  +664.070, Z    +0.000, E1    +5.025, E3 +272935.000}
SPL {X  -159.990, Y  +656.953, Z    +0.000, E1   +13.960, E3 +272936.066}
SPL {X  -159.990, Y  +644.589, Z    +0.000, E1   +29.011, E3 +272939.478}
SPL {X  -159.990, Y  +605.095, Z    +0.000, E1   +49.514, E3 +272964.569}
SPL {X  -159.990, Y  +543.998, Z    +0.000, E1   +54.483, E3 +273030.558}
SPL {X  -159.990, Y  +535.878, Z    +0.000, E1   +54.465, E3 +273042.893}
SPL {X  -159.990, Y  +529.394, Z    +0.000, E1   +54.464, E3 +273052.723}
SPL {X  -159.990, Y  +521.536, Z    +0.000, E1   +54.480, E3 +273064.604}
SPL {X  -159.990, Y  +512.119, Z    +0.000, E1   +54.487, E3 +273078.850}
SPL {X  -159.990, Y  +504.581, Z    +0.000, E1   +54.460, E3 +273090.309}
SPL {X  -159.990, Y  +497.571, Z    +0.000, E1   +54.478, E3 +273100.896}
SPL {X  -159.990, Y  +490.343, Z    +0.000, E1   +54.468, E3 +273111.861}
SPL {X  -159.990, Y  +483.191, Z    +0.000, E1   +54.478, E3 +273122.677}
SPL {X  -159.990, Y  +471.543, Z    +0.000, E1   +55.096, E3 +273136.306}
SPL {X  -159.990, Y  +443.253, Z    +0.000, E1   +59.297, E3 +273147.737}
SPL {X  -159.990, Y  +438.044, Z    +0.000, E1   +58.687, E3 +273158.593}
SPL {X  -159.990, Y  +431.936, Z    +0.000, E1   +57.955, E3 +273171.412}
SPL {X  -159.990, Y  +427.293, Z    +0.000, E1   +56.830, E3 +273185.118}
SPL {X  -159.990, Y  +423.841, Z    +0.000, E1   +55.679, E3 +273197.220}
SPL {X  -159.990, Y  +418.232, Z    +0.000, E1   +55.048, E3 +273209.574}
SPL {X  -159.990, Y  +407.911, Z    +0.000, E1   +54.938, E3 +273225.687}
SPL {X  -159.990, Y  +400.284, Z    +0.000, E1   +54.897, E3 +273237.121}
SPL {X  -159.990, Y  +392.953, Z    +0.000, E1   +54.918, E3 +273248.026}
SPL {X  -159.990, Y  +383.354, Z    +0.000, E1   +54.920, E3 +273262.336}
SPL {X  -159.660, Y  +372.225, Z    +0.000, E1   +54.896, E3 +273279.217}
SPL {X  -158.803, Y  +363.045, Z    +0.000, E1   +54.709, E3 +273293.869}
SPL {X  -157.966, Y  +357.131, Z    +0.000, E1   +54.559, E3 +273303.572}
SPL {X  -156.481, Y  +349.175, Z    +0.000, E1   +54.353, E3 +273316.911}
SPL {X  -154.716, Y  +341.761, Z    +0.000, E1   +53.995, E3 +273329.860}
SPL {X  -152.882, Y  +335.340, Z    +0.000, E1   +53.695, E3 +273341.261}
SPL {X  -151.019, Y  +329.680, Z    +0.000, E1   +53.334, E3 +273351.618}
SPL {X  -148.682, Y  +323.421, Z    +0.000, E1   +52.939, E3 +273363.221}
SPL {X  -145.914, Y  +316.881, Z    +0.000, E1   +52.402, E3 +273375.685}
SPL {X  -142.795, Y  +310.344, Z    +0.000, E1   +51.829, E3 +273388.340}
SPL {X  -132.354, Y  +292.616, Z    +0.000, E1   +44.164, E3 +273486.753}
ENDSPLINE

SPLINE
SPL {X  -150.910, Y  +329.369, Z    +0.000, E1   +29.678, E3 +273559.148}
SPL {X  -156.396, Y  +348.778, Z    +0.000, E1   +21.134, E3 +273570.791}
SPL {X  -158.554, Y  +361.116, Z    +0.000, E1   +14.883, E3 +273575.245}
SPL {X  -159.881, Y  +376.607, Z    +0.000, E1    +5.865, E3 +273578.654}
SPL {X  -159.990, Y  +383.659, Z    +0.000, E1    +1.050, E3 +273579.335}
SPL {X  -159.990, Y  +387.327, Z    +0.000, E1    -2.137, E3 +273579.568}
SPL {X  -159.990, Y  +392.053, Z    +0.000, E1    -7.477, E3 +273580.033}
SPL {X  -159.990, Y  +396.158, Z    +0.000, E1   -12.775, E3 +273580.658}
SPL {X  -159.990, Y  +401.377, Z    +0.000, E1   -19.398, E3 +273581.839}
SPL {X  -159.990, Y  +411.365, Z    +0.000, E1   -30.630, E3 +273585.047}
SPL {X  -159.990, Y  +450.467, Z    +0.000, E1   -50.183, E3 +273608.696}
SPL {X  -159.990, Y  +509.934, Z    +0.000, E1   -54.923, E3 +273671.315}
SPL {X  -159.990, Y  +516.848, Z    +0.000, E1   -54.930, E3 +273681.603}
SPL {X  -159.990, Y  +524.818, Z    +0.000, E1   -54.933, E3 +273693.475}
SPL {X  -159.990, Y  +532.100, Z    +0.000, E1   -54.924, E3 +273704.328}
SPL {X  -159.990, Y  +539.391, Z    +0.000, E1   -54.933, E3 +273715.180}
SPL {X  -159.990, Y  +546.283, Z    +0.000, E1   -54.924, E3 +273725.451}
SPL {X  -159.990, Y  +553.734, Z    +0.000, E1   -54.938, E3 +273736.538}
SPL {X  -159.990, Y  +560.983, Z    +0.000, E1   -54.918, E3 +273747.375}
SPL {X  -159.990, Y  +567.462, Z    +0.000, E1   -54.929, E3 +273757.011}
SPL {X  -159.990, Y  +575.140, Z    +0.000, E1   -54.928, E3 +273768.443}
SPL {X  -159.990, Y  +581.046, Z    +0.000, E1   -54.920, E3 +273777.255}
SPL {X  -159.990, Y  +588.063, Z    +0.000, E1   -54.931, E3 +273787.690}
SPL {X  -159.990, Y  +595.273, Z    +0.000, E1   -54.928, E3 +273798.414}
SPL {X  -159.990, Y  +602.326, Z    +0.000, E1   -54.932, E3 +273808.914}
SPL {X  -159.990, Y  +610.296, Z    +0.000, E1   -54.937, E3 +273820.783}
SPL {X  -159.990, Y  +618.534, Z    +0.000, E1   -54.942, E3 +273833.020}
SPL {X  -159.990, Y  +625.928, Z    +0.000, E1   -54.931, E3 +273844.045}
SPL {X  -159.990, Y  +633.423, Z    +0.000, E1   -54.943, E3 +273855.188}
SPL {X  -159.990, Y  +643.352, Z    +0.000, E1   -54.966, E3 +273869.923}
SPL {X  -159.990, Y  +650.756, Z    +0.000, E1   -54.931, E3 +273880.990}
SPL {X  -159.990, Y  +658.525, Z    +0.000, E1   -54.959, E3 +273892.526}
SPL {X  -159.990, Y  +667.903, Z    +0.000, E1   -54.941, E3 +273906.557}
SPL {X  -159.953, Y  +674.920, Z    +0.000, E1   -54.918, E3 +273917.060}
SPL {X  -159.714, Y  +680.893, Z    +0.000, E1   -54.890, E3 +273926.200}
SPL {X  -159.222, Y  +687.156, Z    +0.000, E1   -54.792, E3 +273936.087}
SPL {X  -158.388, Y  +694.082, Z    +0.000, E1   -54.679, E3 +273947.225}
SPL {X  -157.277, Y  +700.838, Z    +0.000, E1   -54.465, E3 +273958.482}
SPL {X  -156.153, Y  +706.327, Z    +0.000, E1   -54.274, E3 +273967.818}
SPL {X  -154.917, Y  +711.470, Z    +0.000, E1   -54.052, E3 +273976.769}
SPL {X  -153.204, Y  +717.603, Z    +0.000, E1   -53.775, E3 +273987.615}
SPL {X  -151.355, Y  +723.351, Z    +0.000, E1   -53.415, E3 +273998.087}
SPL {X  -149.371, Y  +728.816, Z    +0.000, E1   -53.074, E3 +274008.177}
SPL {X  -147.376, Y  +733.767, Z    +0.000, E1   -52.671, E3 +274017.580}
SPL {X  -145.158, Y  +738.775, Z    +0.000, E1   -52.288, E3 +274027.131}
SPL {X  -142.385, Y  +744.461, Z    +0.000, E1   -51.729, E3 +274038.243}
SPL {X  -132.301, Y  +761.463, Z    +0.000, E1   -45.510, E3 +274115.981}
ENDSPLINE

SPLINE
SPL {X  -145.877, Y  +737.201, Z    +0.000, E1   -34.468, E3 +274199.092}
SPL {X  -152.550, Y  +719.721, Z    +0.000, E1   -27.728, E3 +274214.581}
SPL {X  -157.145, Y  +701.536, Z    +0.000, E1   -19.368, E3 +274224.036}
SPL {X  -159.035, Y  +688.952, Z    +0.000, E1   -12.676, E3 +274228.077}
SPL {X  -159.873, Y  +677.622, Z    +0.000, E1    -6.008, E3 +274230.149}
SPL {X  -159.990, Y  +671.638, Z    +0.000, E1    -1.925, E3 +274230.776}
SPL {X  -159.990, Y  +668.344, Z    +0.000, E1    +0.618, E3 +274230.968}
SPL {X  -159.990, Y  +665.430, Z    +0.000, E1    +3.630, E3 +274231.163}
SPL {X  -159.990, Y  +661.750, Z    +0.000, E1    +7.880, E3 +274231.554}
SPL {X  -159.990, Y  +655.696, Z    +0.000, E1   +15.733, E3 +274232.606}
SPL {X  -159.990, Y  +644.589, Z    +0.000, E1   +29.011, E3 +274235.774}
SPL {X  -159.990, Y  +605.095, Z    +0.000, E1   +49.514, E3 +274260.865}
SPL {X  -159.990, Y  +543.998, Z    +0.000, E1   +54.483, E3 +274326.855}
SPL {X  -159.990, Y  +535.878, Z    +0.000, E1   +54.465, E3 +274339.189}
SPL {X  -159.990, Y  +529.394, Z    +0.000, E1   +54.464, E3 +274349.019}
SPL {X  -159.990, Y  +521.536, Z    +0.000, E1   +54.480, E3 +274360.901}
SPL {X  -159.990, Y  +514.089, Z    +0.000, E1   +54.461, E3 +274372.213}
SPL {X  -159.990, Y  +506.373, Z    +0.000, E1   +54.484, E3 +274383.849}
SPL {X  -159.990, Y  +497.571, Z    +0.000, E1   +54.478, E3 +274397.193}
SPL {X  -159.990, Y  +490.343, Z    +0.000, E1   +54.468, E3 +274408.158}
SPL {X  -159.990, Y  +483.191, Z    +0.000, E1   +54.478, E3 +274418.974}
SPL {X  -159.990, Y  +475.502, Z    +0.000, E1   +54.476, E3 +274430.623}
SPL {X  -159.990, Y  +448.520, Z    +0.000, E1   +58.543, E3 +274442.252}
SPL {X  -159.990, Y  +438.044, Z    +0.000, E1   +58.687, E3 +274454.889}
SPL {X  -159.990, Y  +431.936, Z    +0.000, E1   +57.955, E3 +274467.708}
SPL {X  -159.990, Y  +427.293, Z    +0.000, E1   +56.830, E3 +274481.414}
SPL {X  -159.990, Y  +423.841, Z    +0.000, E1   +55.679, E3 +274493.516}
SPL {X  -159.990, Y  +418.232, Z    +0.000, E1   +55.048, E3 +274505.870}
SPL {X  -159.990, Y  +410.722, Z    +0.000, E1   +54.900, E3 +274517.853}
SPL {X  -159.990, Y  +402.790, Z    +0.000, E1   +54.930, E3 +274529.628}
SPL {X  -159.990, Y  +391.119, Z    +0.000, E1   +54.948, E3 +274547.006}
SPL {X  -159.951, Y  +378.972, Z    +0.000, E1   +54.929, E3 +274565.184}
SPL {X  -159.499, Y  +369.977, Z    +0.000, E1   +54.827, E3 +274579.096}
SPL {X  -158.803, Y  +363.045, Z    +0.000, E1   +54.709, E3 +274590.165}
SPL {X  -157.966, Y  +357.131, Z    +0.000, E1   +54.559, E3 +274599.868}
SPL {X  -156.775, Y  +350.586, Z    +0.000, E1   +54.373, E3 +274610.842}
SPL {X  -155.027, Y  +342.959, Z    +0.000, E1   +54.074, E3 +274624.015}
SPL {X  -153.580, Y  +337.668, Z    +0.000, E1   +53.781, E3 +274633.438}
SPL {X  -151.643, Y  +331.497, Z    +0.000, E1   +53.493, E3 +274644.517}
SPL {X  -149.351, Y  +325.131, Z    +0.000, E1   +53.025, E3 +274656.359}
SPL {X  -147.860, Y  +321.391, Z    +0.000, E1   +52.740, E3 +274663.411}
SPL {X  -145.914, Y  +316.881, Z    +0.000, E1   +52.402, E3 +274671.981}
SPL {X  -142.795, Y  +310.344, Z    +0.000, E1   +51.829, E3 +274684.637}
SPL {X  -132.354, Y  +292.616, Z    +0.000, E1   +44.164, E3 +274783.049}
ENDSPLINE

SPLINE
SPL {X  -150.910, Y  +329.369, Z    +0.000, E1   +29.678, E3 +274855.444}
SPL {X  -156.829, Y  +350.854, Z    +0.000, E1   +20.141, E3 +274867.997}
SPL {X  -159.049, Y  +365.169, Z    +0.000, E1   +12.580, E3 +274872.741}
SPL {X  -159.776, Y  +374.231, Z    +0.000, E1    +7.281, E3 +274874.627}
SPL {X  -159.986, Y  +381.380, Z    +0.000, E1    +2.685, E3 +274875.473}
SPL {X  -159.990, Y  +384.493, Z    +0.000, E1    +0.324, E3 +274875.681}
SPL {X  -159.990, Y  +387.327, Z    +0.000, E1    -2.137, E3 +274875.864}
SPL {X  -159.990, Y  +392.053, Z    +0.000, E1    -7.477, E3 +274876.329}
SPL {X  -159.990, Y  +396.158, Z    +0.000, E1   -12.775, E3 +274876.955}
SPL {X  -159.990, Y  +401.377, Z    +0.000, E1   -19.398, E3 +274878.135}
SPL {X  -159.990, Y  +411.365, Z    +0.000, E1   -30.630, E3 +274881.343}
SPL {X  -159.990, Y  +450.467, Z    +0.000, E1   -50.183, E3 +274904.992}
SPL {X  -159.990, Y  +509.934, Z    +0.000, E1   -54.923, E3 +274967.611}
SPL {X  -159.990, Y  +516.848, Z    +0.000, E1   -54.930, E3 +274977.899}
SPL {X  -159.990, Y  +524.818, Z    +0.000, E1   -54.933, E3 +274989.771}
SPL {X  -159.990, Y  +532.100, Z    +0.000, E1   -54.924, E3 +275000.624}
SPL {X  -159.990, Y  +539.391, Z    +0.000, E1   -54.933, E3 +275011.476}
SPL {X  -159.990, Y  +546.283, Z    +0.000, E1   -54.924, E3 +275021.748}
SPL {X  -159.990, Y  +553.734, Z    +0.000, E1   -54.938, E3 +275032.834}
SPL {X  -159.990, Y  +560.983, Z    +0.000, E1   -54.918, E3 +275043.672}
SPL {X  -159.990, Y  +567.462, Z    +0.000, E1   -54.929, E3 +275053.307}
SPL {X  -159.990, Y  +575.140, Z    +0.000, E1   -54.928, E3 +275064.739}
SPL {X  -159.990, Y  +581.046, Z    +0.000, E1   -54.920, E3 +275073.551}
SPL {X  -159.990, Y  +588.063, Z    +0.000, E1   -54.931, E3 +275083.986}
SPL {X  -159.990, Y  +595.273, Z    +0.000, E1   -54.928, E3 +275094.710}
SPL {X  -159.990, Y  +602.326, Z    +0.000, E1   -54.932, E3 +275105.210}
SPL {X  -159.990, Y  +610.296, Z    +0.000, E1   -54.937, E3 +275117.080}
SPL {X  -159.990, Y  +618.534, Z    +0.000, E1   -54.942, E3 +275129.317}
SPL {X  -159.990, Y  +628.178, Z    +0.000, E1   -54.959, E3 +275143.648}
SPL {X  -159.990, Y  +638.304, Z    +0.000, E1   -54.952, E3 +275158.737}
SPL {X  -159.990, Y  +645.976, Z    +0.000, E1   -54.934, E3 +275170.171}
SPL {X  -159.990, Y  +650.756, Z    +0.000, E1   -54.931, E3 +275177.286}
SPL {X  -159.990, Y  +658.525, Z    +0.000, E1   -54.959, E3 +275188.822}
SPL {X  -159.990, Y  +667.903, Z    +0.000, E1   -54.941, E3 +275202.853}
SPL {X  -159.827, Y  +678.718, Z    +0.000, E1   -54.950, E3 +275219.072}
SPL {X  -159.222, Y  +687.156, Z    +0.000, E1   -54.792, E3 +275232.383}
SPL {X  -158.388, Y  +694.082, Z    +0.000, E1   -54.679, E3 +275243.521}
SPL {X  -157.277, Y  +700.838, Z    +0.000, E1   -54.465, E3 +275254.778}
SPL {X  -156.153, Y  +706.327, Z    +0.000, E1   -54.274, E3 +275264.114}
SPL {X  -154.917, Y  +711.470, Z    +0.000, E1   -54.052, E3 +275273.066}
SPL {X  -153.204, Y  +717.603, Z    +0.000, E1   -53.775, E3 +275283.912}
SPL {X  -151.355, Y  +723.351, Z    +0.000, E1   -53.415, E3 +275294.383}
SPL {X  -149.371, Y  +728.816, Z    +0.000, E1   -53.074, E3 +275304.474}
SPL {X  -146.631, Y  +735.501, Z    +0.000, E1   -52.568, E3 +275317.134}
SPL {X  -144.428, Y  +740.329, Z    +0.000, E1   -52.109, E3 +275326.488}
SPL {X  -142.385, Y  +744.461, Z    +0.000, E1   -51.729, E3 +275334.539}
SPL {X  -132.301, Y  +761.463, Z    +0.000, E1   -45.510, E3 +275412.278}
ENDSPLINE

SPLINE
SPL {X  -145.877, Y  +737.201, Z    +0.000, E1   -34.468, E3 +275495.388}
SPL {X  -152.550, Y  +719.721, Z    +0.000, E1   -27.728, E3 +275510.878}
SPL {X  -157.145, Y  +701.536, Z    +0.000, E1   -19.368, E3 +275520.332}
SPL {X  -159.035, Y  +688.952, Z    +0.000, E1   -12.676, E3 +275524.373}
SPL {X  -159.756, Y  +680.154, Z    +0.000, E1    -7.520, E3 +275526.100}
SPL {X  -159.986, Y  +672.560, Z    +0.000, E1    -2.636, E3 +275526.998}
SPL {X  -159.990, Y  +668.344, Z    +0.000, E1    +0.618, E3 +275527.264}
SPL {X  -159.990, Y  +664.070, Z    +0.000, E1    +5.025, E3 +275527.592}
SPL {X  -159.990, Y  +656.953, Z    +0.000, E1   +13.960, E3 +275528.659}
SPL {X  -159.990, Y  +644.589, Z    +0.000, E1   +29.011, E3 +275532.070}
SPL {X  -159.990, Y  +605.095, Z    +0.000, E1   +49.514, E3 +275557.161}
SPL {X  -159.990, Y  +543.998, Z    +0.000, E1   +54.483, E3 +275623.151}
SPL {X  -159.990, Y  +535.878, Z    +0.000, E1   +54.465, E3 +275635.486}
SPL {X  -159.990, Y  +529.394, Z    +0.000, E1   +54.464, E3 +275645.315}
SPL {X  -159.990, Y  +521.536, Z    +0.000, E1   +54.480, E3 +275657.197}
SPL {X  -159.990, Y  +514.089, Z    +0.000, E1   +54.461, E3 +275668.509}
SPL {X  -159.990, Y  +506.373, Z    +0.000, E1   +54.484, E3 +275680.146}
SPL {X  -159.990, Y  +497.571, Z    +0.000, E1   +54.478, E3 +275693.489}
SPL {X  -159.990, Y  +490.343, Z    +0.000, E1   +54.468, E3 +275704.454}
SPL {X  -159.990, Y  +483.191, Z    +0.000, E1   +54.478, E3 +275715.270}
SPL {X  -159.990, Y  +475.502, Z    +0.000, E1   +54.476, E3 +275726.919}
SPL {X  -159.990, Y  +448.520, Z    +0.000, E1   +58.543, E3 +275738.548}
SPL {X  -159.990, Y  +438.044, Z    +0.000, E1   +58.687, E3 +275751.185}
SPL {X  -159.990, Y  +431.936, Z    +0.000, E1   +57.955, E3 +275764.005}
SPL {X  -159.990, Y  +427.860, Z    +0.000, E1   +57.091, E3 +275775.068}
SPL {X  -159.990, Y  +424.653, Z    +0.000, E1   +55.901, E3 +275787.374}
SPL {X  -159.990, Y  +419.589, Z    +0.000, E1   +55.096, E3 +275799.737}
SPL {X  -159.990, Y  +412.636, Z    +0.000, E1   +54.925, E3 +275811.249}
SPL {X  -159.990, Y  +405.235, Z    +0.000, E1   +54.902, E3 +275822.319}
SPL {X  -159.990, Y  +400.284, Z    +0.000, E1   +54.897, E3 +275829.714}
SPL {X  -159.990, Y  +392.953, Z    +0.000, E1   +54.918, E3 +275840.618}
SPL {X  -159.990, Y  +383.354, Z    +0.000, E1   +54.920, E3 +275854.928}
SPL {X  -159.860, Y  +376.053, Z    +0.000, E1   +54.872, E3 +275865.988}
SPL {X  -159.499, Y  +369.977, Z    +0.000, E1   +54.827, E3 +275875.393}
SPL {X  -158.803, Y  +363.045, Z    +0.000, E1   +54.709, E3 +275886.461}
SPL {X  -157.732, Y  +355.717, Z    +0.000, E1   +54.540, E3 +275898.484}
SPL {X  -156.235, Y  +348.039, Z    +0.000, E1   +54.281, E3 +275911.495}
SPL {X  -154.264, Y  +340.082, Z    +0.000, E1   +53.947, E3 +275925.372}
SPL {X  -151.643, Y  +331.497, Z    +0.000, E1   +53.493, E3 +275940.813}
SPL {X  -148.682, Y  +323.421, Z    +0.000, E1   +52.939, E3 +275955.813}
SPL {X  -145.914, Y  +316.881, Z    +0.000, E1   +52.402, E3 +275968.277}
SPL {X  -143.679, Y  +312.121, Z    +0.000, E1   +51.954, E3 +275977.522}
SPL {X  -141.812, Y  +308.430, Z    +0.000, E1   +51.590, E3 +275984.754}
SPL {X  -132.354, Y  +292.616, Z    +0.000, E1   +44.164, E3 +276079.345}
ENDSPLINE

SPLINE
SPL {X  -150.910, Y  +329.369, Z    +0.000, E1   +29.678, E3 +276151.741}
SPL {X  -156.829, Y  +350.854, Z    +0.000, E1   +20.141, E3 +276164.293}
SPL {X  -159.049, Y  +365.169, Z    +0.000, E1   +12.580, E3 +276169.038}
SPL {X  -159.776, Y  +374.231, Z    +0.000, E1    +7.281, E3 +276170.924}
SPL {X  -159.986, Y  +381.380, Z    +0.000, E1    +2.685, E3 +276171.770}
SPL {X  -159.990, Y  +384.493, Z    +0.000, E1    +0.324, E3 +276171.978}
SPL {X  -159.990, Y  +387.327, Z    +0.000, E1    -2.137, E3 +276172.160}
SPL {X  -159.990, Y  +392.053, Z    +0.000, E1    -7.477, E3 +276172.625}
SPL {X  -159.990, Y  +396.158, Z    +0.000, E1   -12.775, E3 +276173.251}
SPL {X  -159.990, Y  +401.377, Z    +0.000, E1   -19.398, E3 +276174.431}
SPL {X  -159.990, Y  +411.365, Z    +0.000, E1   -30.630, E3 +276177.640}
SPL {X  -159.990, Y  +450.467, Z    +0.000, E1   -50.183, E3 +276201.288}
SPL {X  -159.990, Y  +509.934, Z    +0.000, E1   -54.923, E3 +276263.907}
SPL {X  -159.990, Y  +516.848, Z    +0.000, E1   -54.930, E3 +276274.195}
SPL {X  -159.990, Y  +524.818, Z    +0.000, E1   -54.933, E3 +276286.067}
SPL {X  -159.990, Y  +532.100, Z    +0.000, E1   -54.924, E3 +276296.920}
SPL {X  -159.990, Y  +539.391, Z    +0.000, E1   -54.933, E3 +276307.772}
SPL {X  -159.990, Y  +546.283, Z    +0.000, E1   -54.924, E3 +276318.044}
SPL {X  -159.990, Y  +553.734, Z    +0.000, E1   -54.938, E3 +276329.131}
SPL {X  -159.990, Y  +564.956, Z    +0.000, E1   -54.973, E3 +276345.802}
SPL {X  -159.990, Y  +575.140, Z    +0.000, E1   -54.928, E3 +276361.035}
SPL {X  -159.990, Y  +581.046, Z    +0.000, E1   -54.920, E3 +276369.848}
SPL {X  -159.990, Y  +588.063, Z    +0.000, E1   -54.931, E3 +276380.283}
SPL {X  -159.990, Y  +595.273, Z    +0.000, E1   -54.928, E3 +276391.006}
SPL {X  -159.990, Y  +602.326, Z    +0.000, E1   -54.932, E3 +276401.507}
SPL {X  -159.990, Y  +610.296, Z    +0.000, E1   -54.937, E3 +276413.376}
SPL {X  -159.990, Y  +618.534, Z    +0.000, E1   -54.942, E3 +276425.613}
SPL {X  -159.990, Y  +625.928, Z    +0.000, E1   -54.931, E3 +276436.638}
SPL {X  -159.990, Y  +633.423, Z    +0.000, E1   -54.943, E3 +276447.780}
SPL {X  -159.990, Y  +640.333, Z    +0.000, E1   -54.927, E3 +276458.095}
SPL {X  -159.990, Y  +648.272, Z    +0.000, E1   -54.961, E3 +276469.842}
SPL {X  -159.990, Y  +655.990, Z    +0.000, E1   -54.930, E3 +276481.390}
SPL {X  -159.990, Y  +665.734, Z    +0.000, E1   -54.984, E3 +276495.841}
SPL {X  -159.953, Y  +674.920, Z    +0.000, E1   -54.918, E3 +276509.652}
SPL {X  -159.714, Y  +680.893, Z    +0.000, E1   -54.890, E3 +276518.792}
SPL {X  -159.222, Y  +687.156, Z    +0.000, E1   -54.792, E3 +276528.680}
SPL {X  -158.388, Y  +694.082, Z    +0.000, E1   -54.679, E3 +276539.817}
SPL {X  -157.277, Y  +700.838, Z    +0.000, E1   -54.465, E3 +276551.075}
SPL {X  -156.153, Y  +706.327, Z    +0.000, E1   -54.274, E3 +276560.411}
SPL {X  -154.505, Y  +713.032, Z    +0.000, E1   -54.006, E3 +276572.072}
SPL {X  -152.808, Y  +718.896, Z    +0.000, E1   -53.679, E3 +276582.569}
SPL {X  -150.773, Y  +725.019, Z    +0.000, E1   -53.343, E3 +276593.701}
SPL {X  -148.029, Y  +732.198, Z    +0.000, E1   -52.831, E3 +276607.138}
SPL {X  -145.158, Y  +738.775, Z    +0.000, E1   -52.288, E3 +276619.723}
SPL {X  -142.385, Y  +744.461, Z    +0.000, E1   -51.729, E3 +276630.835}
SPL {X  -132.301, Y  +761.463, Z    +0.000, E1   -45.510, E3 +276708.574}
ENDSPLINE

SPLINE
SPL {X  -145.877, Y  +737.201, Z    +0.000, E1   -34.468, E3 +276791.685}
SPL {X  -152.550, Y  +719.721, Z    +0.000, E1   -27.728, E3 +276807.174}
SPL {X  -157.145, Y  +701.536, Z    +0.000, E1   -19.368, E3 +276816.629}
SPL {X  -159.035, Y  +688.952, Z    +0.000, E1   -12.676, E3 +276820.670}
SPL {X  -159.756, Y  +680.154, Z    +0.000, E1    -7.520, E3 +276822.396}
SPL {X  -159.986, Y  +672.560, Z    +0.000, E1    -2.636, E3 +276823.294}
SPL {X  -159.990, Y  +668.344, Z    +0.000, E1    +0.618, E3 +276823.560}
SPL {X  -159.990, Y  +664.070, Z    +0.000, E1    +5.025, E3 +276823.889}
SPL {X  -159.990, Y  +656.953, Z    +0.000, E1   +13.960, E3 +276824.955}
SPL {X  -159.990, Y  +644.589, Z    +0.000, E1   +29.011, E3 +276828.367}
SPL {X  -159.990, Y  +605.095, Z    +0.000, E1   +49.514, E3 +276853.457}
SPL {X  -159.990, Y  +543.998, Z    +0.000, E1   +54.483, E3 +276919.447}
SPL {X  -159.990, Y  +535.878, Z    +0.000, E1   +54.465, E3 +276931.782}
SPL {X  -159.990, Y  +529.394, Z    +0.000, E1   +54.464, E3 +276941.612}
SPL {X  -159.990, Y  +521.536, Z    +0.000, E1   +54.480, E3 +276953.493}
SPL {X  -159.990, Y  +514.089, Z    +0.000, E1   +54.461, E3 +276964.806}
SPL {X  -159.990, Y  +506.373, Z    +0.000, E1   +54.484, E3 +276976.442}
SPL {X  -159.990, Y  +497.571, Z    +0.000, E1   +54.478, E3 +276989.785}
SPL {X  -159.990, Y  +490.343, Z    +0.000, E1   +54.468, E3 +277000.750}
SPL {X  -159.990, Y  +483.191, Z    +0.000, E1   +54.478, E3 +277011.566}
SPL {X  -159.990, Y  +471.543, Z    +0.000, E1   +55.096, E3 +277025.194}
SPL {X  -159.990, Y  +443.253, Z    +0.000, E1   +59.297, E3 +277036.626}
SPL {X  -159.990, Y  +438.044, Z    +0.000, E1   +58.687, E3 +277047.481}
SPL {X  -159.990, Y  +431.936, Z    +0.000, E1   +57.955, E3 +277060.301}
SPL {X  -159.990, Y  +427.860, Z    +0.000, E1   +57.091, E3 +277071.365}
SPL {X  -159.990, Y  +424.653, Z    +0.000, E1   +55.901, E3 +277083.670}
SPL {X  -159.990, Y  +418.232, Z    +0.000, E1   +55.048, E3 +277098.463}
SPL {X  -159.990, Y  +410.722, Z    +0.000, E1   +54.900, E3 +277110.446}
SPL {X  -159.990, Y  +402.790, Z    +0.000, E1   +54.930, E3 +277122.221}
SPL {X  -159.990, Y  +391.119, Z    +0.000, E1   +54.948, E3 +277139.598}
SPL {X  -159.951, Y  +378.972, Z    +0.000, E1   +54.929, E3 +277157.777}
SPL {X  -159.499, Y  +369.977, Z    +0.000, E1   +54.827, E3 +277171.689}
SPL {X  -158.803, Y  +363.045, Z    +0.000, E1   +54.709, E3 +277182.758}
SPL {X  -157.966, Y  +357.131, Z    +0.000, E1   +54.559, E3 +277192.461}
SPL {X  -156.775, Y  +350.586, Z    +0.000, E1   +54.373, E3 +277203.435}
SPL {X  -155.027, Y  +342.959, Z    +0.000, E1   +54.074, E3 +277216.607}
SPL {X  -152.882, Y  +335.340, Z    +0.000, E1   +53.695, E3 +277230.150}
SPL {X  -151.019, Y  +329.680, Z    +0.000, E1   +53.334, E3 +277240.507}
SPL {X  -149.351, Y  +325.131, Z    +0.000, E1   +53.025, E3 +277248.951}
SPL {X  -147.860, Y  +321.391, Z    +0.000, E1   +52.740, E3 +277256.004}
SPL {X  -145.914, Y  +316.881, Z    +0.000, E1   +52.402, E3 +277264.574}
SPL {X  -142.795, Y  +310.344, Z    +0.000, E1   +51.829, E3 +277277.229}
SPL {X  -132.354, Y  +292.616, Z    +0.000, E1   +44.164, E3 +277375.642}
ENDSPLINE

SPLINE
SPL {X  -150.910, Y  +329.369, Z    +0.000, E1   +29.678, E3 +277448.037}
SPL {X  -156.396, Y  +348.778, Z    +0.000, E1   +21.134, E3 +277459.680}
SPL {X  -158.554, Y  +361.116, Z    +0.000, E1   +14.883, E3 +277464.134}
SPL {X  -159.881, Y  +376.607, Z    +0.000, E1    +5.865, E3 +277467.543}
SPL {X  -159.990, Y  +383.659, Z    +0.000, E1    +1.050, E3 +277468.224}
SPL {X  -159.990, Y  +387.327, Z    +0.000, E1    -2.137, E3 +277468.457}
SPL {X  -159.990, Y  +390.622, Z    +0.000, E1    -5.876, E3 +277468.750}
SPL {X  -159.990, Y  +394.493, Z    +0.000, E1   -10.512, E3 +277469.273}
SPL {X  -159.990, Y  +401.377, Z    +0.000, E1   -19.398, E3 +277470.727}
SPL {X  -159.990, Y  +411.365, Z    +0.000, E1   -30.630, E3 +277473.936}
SPL {X  -159.990, Y  +450.467, Z    +0.000, E1   -50.183, E3 +277497.585}
SPL {X  -159.990, Y  +509.934, Z    +0.000, E1   -54.923, E3 +277560.204}
SPL {X  -159.990, Y  +516.848, Z    +0.000, E1   -54.930, E3 +277570.492}
SPL {X  -159.990, Y  +524.818, Z    +0.000, E1   -54.933, E3 +277582.364}
SPL {X  -159.990, Y  +532.100, Z    +0.000, E1   -54.924, E3 +277593.217}
SPL {X  -159.990, Y  +539.391, Z    +0.000, E1   -54.933, E3 +277604.069}
SPL {X  -159.990, Y  +546.283, Z    +0.000, E1   -54.924, E3 +277614.340}
SPL {X  -159.990, Y  +553.734, Z    +0.000, E1   -54.938, E3 +277625.427}
SPL {X  -159.990, Y  +564.956, Z    +0.000, E1   -54.973, E3 +277642.098}
SPL {X  -159.990, Y  +577.902, Z    +0.000, E1   -54.969, E3 +277661.388}
SPL {X  -159.990, Y  +588.063, Z    +0.000, E1   -54.931, E3 +277676.579}
SPL {X  -159.990, Y  +595.273, Z    +0.000, E1   -54.928, E3 +277687.302}
SPL {X  -159.990, Y  +602.326, Z    +0.000, E1   -54.932, E3 +277697.803}
SPL {X  -159.990, Y  +610.296, Z    +0.000, E1   -54.937, E3 +277709.672}
SPL {X  -159.990, Y  +618.534, Z    +0.000, E1   -54.942, E3 +277721.909}
SPL {X  -159.990, Y  +628.178, Z    +0.000, E1   -54.959, E3 +277736.240}
SPL {X  -159.990, Y  +638.304, Z    +0.000, E1   -54.952, E3 +277751.329}
SPL {X  -159.990, Y  +648.272, Z    +0.000, E1   -54.961, E3 +277766.138}
SPL {X  -159.990, Y  +655.990, Z    +0.000, E1   -54.930, E3 +277777.686}
SPL {X  -159.990, Y  +665.734, Z    +0.000, E1   -54.984, E3 +277792.137}
SPL {X  -159.827, Y  +678.718, Z    +0.000, E1   -54.950, E3 +277811.665}
SPL {X  -159.222, Y  +687.156, Z    +0.000, E1   -54.792, E3 +277824.976}
SPL {X  -158.388, Y  +694.082, Z    +0.000, E1   -54.679, E3 +277836.114}
SPL {X  -157.277, Y  +700.838, Z    +0.000, E1   -54.465, E3 +277847.371}
SPL {X  -156.153, Y  +706.327, Z    +0.000, E1   -54.274, E3 +277856.707}
SPL {X  -154.917, Y  +711.470, Z    +0.000, E1   -54.052, E3 +277865.658}
SPL {X  -153.204, Y  +717.603, Z    +0.000, E1   -53.775, E3 +277876.504}
SPL {X  -151.355, Y  +723.351, Z    +0.000, E1   -53.415, E3 +277886.976}
SPL {X  -149.371, Y  +728.816, Z    +0.000, E1   -53.074, E3 +277897.066}
SPL {X  -147.376, Y  +733.767, Z    +0.000, E1   -52.671, E3 +277906.468}
SPL {X  -145.158, Y  +738.775, Z    +0.000, E1   -52.288, E3 +277916.020}
SPL {X  -142.385, Y  +744.461, Z    +0.000, E1   -51.729, E3 +277927.131}
SPL {X  -132.301, Y  +761.463, Z    +0.000, E1   -45.510, E3 +278004.870}
ENDSPLINE

SPLINE
SPL {X  -145.877, Y  +737.201, Z    +0.000, E1   -34.468, E3 +278087.981}
SPL {X  -152.550, Y  +719.721, Z    +0.000, E1   -27.728, E3 +278103.470}
SPL {X  -157.145, Y  +701.536, Z    +0.000, E1   -19.368, E3 +278112.925}
SPL {X  -159.035, Y  +688.952, Z    +0.000, E1   -12.676, E3 +278116.966}
SPL {X  -159.756, Y  +680.154, Z    +0.000, E1    -7.520, E3 +278118.692}
SPL {X  -159.986, Y  +672.560, Z    +0.000, E1    -2.636, E3 +278119.590}
SPL {X  -159.990, Y  +668.344, Z    +0.000, E1    +0.618, E3 +278119.857}
SPL {X  -159.990, Y  +664.070, Z    +0.000, E1    +5.025, E3 +278120.185}
SPL {X  -159.990, Y  +656.953, Z    +0.000, E1   +13.960, E3 +278121.251}
SPL {X  -159.990, Y  +644.589, Z    +0.000, E1   +29.011, E3 +278124.663}
SPL {X  -159.990, Y  +605.095, Z    +0.000, E1   +49.514, E3 +278149.754}
SPL {X  -159.990, Y  +546.155, Z    +0.000, E1   +54.461, E3 +278212.512}
SPL {X  -159.990, Y  +537.700, Z    +0.000, E1   +54.492, E3 +278225.276}
SPL {X  -159.990, Y  +529.394, Z    +0.000, E1   +54.464, E3 +278237.908}
SPL {X  -159.990, Y  +521.536, Z    +0.000, E1   +54.480, E3 +278249.790}
SPL {X  -159.990, Y  +514.089, Z    +0.000, E1   +54.461, E3 +278261.102}
SPL {X  -159.990, Y  +506.373, Z    +0.000, E1   +54.484, E3 +278272.738}
SPL {X  -159.990, Y  +497.571, Z    +0.000, E1   +54.478, E3 +278286.081}
SPL {X  -159.990, Y  +490.343, Z    +0.000, E1   +54.468, E3 +278297.046}
SPL {X  -159.990, Y  +483.191, Z    +0.000, E1   +54.478, E3 +278307.863}
SPL {X  -159.990, Y  +475.502, Z    +0.000, E1   +54.476, E3 +278319.512}
SPL {X  -159.990, Y  +448.520, Z    +0.000, E1   +58.543, E3 +278331.141}
SPL {X  -159.990, Y  +438.044, Z    +0.000, E1   +58.687, E3 +278343.778}
SPL {X  -159.990, Y  +431.936, Z    +0.000, E1   +57.955, E3 +278356.597}
SPL {X  -159.990, Y  +427.860, Z    +0.000, E1   +57.091, E3 +278367.661}
SPL {X  -159.990, Y  +424.653, Z    +0.000, E1   +55.901, E3 +278379.966}
SPL {X  -159.990, Y  +418.232, Z    +0.000, E1   +55.048, E3 +278394.759}
SPL {X  -159.990, Y  +410.722, Z    +0.000, E1   +54.900, E3 +278406.742}
SPL {X  -159.990, Y  +402.790, Z    +0.000, E1   +54.930, E3 +278418.517}
SPL {X  -159.990, Y  +392.953, Z    +0.000, E1   +54.918, E3 +278433.211}
SPL {X  -159.990, Y  +383.354, Z    +0.000, E1   +54.920, E3 +278447.521}
SPL {X  -159.860, Y  +376.053, Z    +0.000, E1   +54.872, E3 +278458.581}
SPL {X  -159.499, Y  +369.977, Z    +0.000, E1   +54.827, E3 +278467.985}
SPL {X  -158.803, Y  +363.045, Z    +0.000, E1   +54.709, E3 +278479.054}
SPL {X  -157.732, Y  +355.717, Z    +0.000, E1   +54.540, E3 +278491.076}
SPL {X  -156.235, Y  +348.039, Z    +0.000, E1   +54.281, E3 +278504.088}
SPL {X  -154.716, Y  +341.761, Z    +0.000, E1   +53.995, E3 +278515.045}
SPL {X  -152.882, Y  +335.340, Z    +0.000, E1   +53.695, E3 +278526.446}
SPL {X  -151.019, Y  +329.680, Z    +0.000, E1   +53.334, E3 +278536.803}
SPL {X  -149.351, Y  +325.131, Z    +0.000, E1   +53.025, E3 +278545.247}
SPL {X  -147.860, Y  +321.391, Z    +0.000, E1   +52.740, E3 +278552.300}
SPL {X  -145.914, Y  +316.881, Z    +0.000, E1   +52.402, E3 +278560.870}
SPL {X  -142.795, Y  +310.344, Z    +0.000, E1   +51.829, E3 +278573.526}
SPL {X  -132.354, Y  +292.616, Z    +0.000, E1   +44.164, E3 +278671.938}
ENDSPLINE

SPLINE
SPL {X  -150.910, Y  +329.369, Z    +0.000, E1   +29.678, E3 +278744.333}
SPL {X  -156.829, Y  +350.854, Z    +0.000, E1   +20.141, E3 +278756.886}
SPL {X  -159.049, Y  +365.169, Z    +0.000, E1   +12.580, E3 +278761.630}
SPL {X  -159.776, Y  +374.231, Z    +0.000, E1    +7.281, E3 +278763.516}
SPL {X  -159.986, Y  +381.380, Z    +0.000, E1    +2.685, E3 +278764.362}
SPL {X  -159.990, Y  +384.493, Z    +0.000, E1    +0.324, E3 +278764.570}
SPL {X  -159.990, Y  +387.327, Z    +0.000, E1    -2.137, E3 +278764.753}
SPL {X  -159.990, Y  +392.053, Z    +0.000, E1    -7.477, E3 +278765.218}
SPL {X  -159.990, Y  +396.158, Z    +0.000, E1   -12.775, E3 +278765.844}
SPL {X  -159.990, Y  +401.377, Z    +0.000, E1   -19.398, E3 +278767.024}
SPL {X  -159.990, Y  +411.365, Z    +0.000, E1   -30.630, E3 +278770.232}
SPL {X  -159.990, Y  +450.467, Z    +0.000, E1   -50.183, E3 +278793.881}
SPL {X  -159.990, Y  +509.934, Z    +0.000, E1   -54.923, E3 +278856.500}
SPL {X  -159.990, Y  +516.848, Z    +0.000, E1   -54.930, E3 +278866.788}
SPL {X  -159.990, Y  +524.818, Z    +0.000, E1   -54.933, E3 +278878.660}
SPL {X  -159.990, Y  +532.100, Z    +0.000, E1   -54.924, E3 +278889.513}
SPL {X  -159.990, Y  +539.391, Z    +0.000, E1   -54.933, E3 +278900.365}
SPL {X  -159.990, Y  +546.283, Z    +0.000, E1   -54.924, E3 +278910.637}
SPL {X  -159.990, Y  +553.734, Z    +0.000, E1   -54.938, E3 +278921.723}
SPL {X  -159.990, Y  +560.983, Z    +0.000, E1   -54.918, E3 +278932.561}
SPL {X  -159.990, Y  +567.462, Z    +0.000, E1   -54.929, E3 +278942.196}
SPL {X  -159.990, Y  +575.140, Z    +0.000, E1   -54.928, E3 +278953.628}
SPL {X  -159.990, Y  +581.046, Z    +0.000, E1   -54.920, E3 +278962.440}
SPL {X  -159.990, Y  +588.063, Z    +0.000, E1   -54.931, E3 +278972.875}
SPL {X  -159.990, Y  +595.273, Z    +0.000, E1   -54.928, E3 +278983.599}
SPL {X  -159.990, Y  +602.326, Z    +0.000, E1   -54.932, E3 +278994.099}
SPL {X  -159.990, Y  +610.296, Z    +0.000, E1   -54.937, E3 +279005.969}
SPL {X  -159.990, Y  +618.534, Z    +0.000, E1   -54.942, E3 +279018.206}
SPL {X  -159.990, Y  +625.928, Z    +0.000, E1   -54.931, E3 +279029.231}
SPL {X  -159.990, Y  +633.423, Z    +0.000, E1   -54.943, E3 +279040.373}
SPL {X  -159.990, Y  +643.352, Z    +0.000, E1   -54.966, E3 +279055.108}
SPL {X  -159.990, Y  +650.756, Z    +0.000, E1   -54.931, E3 +279066.175}
SPL {X  -159.990, Y  +658.525, Z    +0.000, E1   -54.959, E3 +279077.711}
SPL {X  -159.990, Y  +667.903, Z    +0.000, E1   -54.941, E3 +279091.742}
SPL {X  -159.953, Y  +674.920, Z    +0.000, E1   -54.918, E3 +279102.245}
SPL {X  -159.714, Y  +680.893, Z    +0.000, E1   -54.890, E3 +279111.385}
SPL {X  -159.222, Y  +687.156, Z    +0.000, E1   -54.792, E3 +279121.272}
SPL {X  -158.388, Y  +694.082, Z    +0.000, E1   -54.679, E3 +279132.410}
SPL {X  -157.277, Y  +700.838, Z    +0.000, E1   -54.465, E3 +279143.667}
SPL {X  -156.153, Y  +706.327, Z    +0.000, E1   -54.274, E3 +279153.003}
SPL {X  -154.917, Y  +711.470, Z    +0.000, E1   -54.052, E3 +279161.954}
SPL {X  -153.204, Y  +717.603, Z    +0.000, E1   -53.775, E3 +279172.801}
SPL {X  -151.355, Y  +723.351, Z    +0.000, E1   -53.415, E3 +279183.272}
SPL {X  -149.371, Y  +728.816, Z    +0.000, E1   -53.074, E3 +279193.363}
SPL {X  -146.631, Y  +735.501, Z    +0.000, E1   -52.568, E3 +279206.023}
SPL {X  -144.428, Y  +740.329, Z    +0.000, E1   -52.109, E3 +279215.377}
SPL {X  -142.385, Y  +744.461, Z    +0.000, E1   -51.729, E3 +279223.428}
SPL {X  -132.301, Y  +761.463, Z    +0.000, E1   -45.510, E3 +279301.166}
ENDSPLINE

SPLINE
SPL {X  -145.877, Y  +737.201, Z    +0.000, E1   -34.468, E3 +279384.277}
SPL {X  -152.550, Y  +719.721, Z    +0.000, E1   -27.728, E3 +279399.766}
SPL {X  -157.145, Y  +701.536, Z    +0.000, E1   -19.368, E3 +279409.221}
SPL {X  -159.035, Y  +688.952, Z    +0.000, E1   -12.676, E3 +279413.262}
SPL {X  -159.756, Y  +680.154, Z    +0.000, E1    -7.520, E3 +279414.989}
SPL {X  -159.986, Y  +672.560, Z    +0.000, E1    -2.636, E3 +279415.887}
SPL {X  -159.990, Y  +668.344, Z    +0.000, E1    +0.618, E3 +279416.153}
SPL {X  -159.990, Y  +665.430, Z    +0.000, E1    +3.630, E3 +279416.348}
SPL {X  -159.990, Y  +661.750, Z    +0.000, E1    +7.880, E3 +279416.739}
SPL {X  -159.990, Y  +657.656, Z    +0.000, E1   +13.276, E3 +279417.384}
SPL {X  -159.990, Y  +652.023, Z    +0.000, E1   +20.449, E3 +279418.672}
SPL {X  -159.990, Y  +641.935, Z    +0.000, E1   +31.848, E3 +279421.844}
SPL {X  -159.990, Y  +605.095, Z    +0.000, E1   +49.514, E3 +279446.050}
SPL {X  -159.990, Y  +546.155, Z    +0.000, E1   +54.461, E3 +279508.809}
SPL {X  -159.990, Y  +537.700, Z    +0.000, E1   +54.492, E3 +279521.572}
SPL {X  -159.990, Y  +529.394, Z    +0.000, E1   +54.464, E3 +279534.204}
SPL {X  -159.990, Y  +521.536, Z    +0.000, E1   +54.480, E3 +279546.086}
SPL {X  -159.990, Y  +512.119, Z    +0.000, E1   +54.487, E3 +279560.332}
SPL {X  -159.990, Y  +504.581, Z    +0.000, E1   +54.460, E3 +279571.791}
SPL {X  -159.990, Y  +497.571, Z    +0.000, E1   +54.478, E3 +279582.378}
SPL {X  -159.990, Y  +490.343, Z    +0.000, E1   +54.468, E3 +279593.343}
SPL {X  -159.990, Y  +483.191, Z    +0.000, E1   +54.478, E3 +279604.159}
SPL {X  -159.990, Y  +475.502, Z    +0.000, E1   +54.476, E3 +279615.808}
SPL {X  -159.990, Y  +448.520, Z    +0.000, E1   +58.543, E3 +279627.437}
SPL {X  -159.990, Y  +438.044, Z    +0.000, E1   +58.687, E3 +279640.074}
SPL {X  -159.990, Y  +431.936, Z    +0.000, E1   +57.955, E3 +279652.894}
SPL {X  -159.990, Y  +427.293, Z    +0.000, E1   +56.830, E3 +279666.600}
SPL {X  -159.990, Y  +423.841, Z    +0.000, E1   +55.679, E3 +279678.701}
SPL {X  -159.990, Y  +418.232, Z    +0.000, E1   +55.048, E3 +279691.055}
SPL {X  -159.990, Y  +410.722, Z    +0.000, E1   +54.900, E3 +279703.038}
SPL {X  -159.990, Y  +402.790, Z    +0.000, E1   +54.930, E3 +279714.813}
SPL {X  -159.990, Y  +391.119, Z    +0.000, E1   +54.948, E3 +279732.191}
SPL {X  -159.951, Y  +378.972, Z    +0.000, E1   +54.929, E3 +279750.369}
SPL {X  -159.499, Y  +369.977, Z    +0.000, E1   +54.827, E3 +279764.282}
SPL {X  -158.803, Y  +363.045, Z    +0.000, E1   +54.709, E3 +279775.350}
SPL {X  -157.966, Y  +357.131, Z    +0.000, E1   +54.559, E3 +279785.053}
SPL {X  -156.775, Y  +350.586, Z    +0.000, E1   +54.373, E3 +279796.027}
SPL {X  -155.027, Y  +342.959, Z    +0.000, E1   +54.074, E3 +279809.200}
SPL {X  -153.580, Y  +337.668, Z    +0.000, E1   +53.781, E3 +279818.623}
SPL {X  -151.643, Y  +331.497, Z    +0.000, E1   +53.493, E3 +279829.702}
SPL {X  -148.682, Y  +323.421, Z    +0.000, E1   +52.939, E3 +279844.702}
SPL {X  -145.914, Y  +316.881, Z    +0.000, E1   +52.402, E3 +279857.166}
SPL {X  -142.795, Y  +310.344, Z    +0.000, E1   +51.829, E3 +279869.822}
SPL {X  -132.354, Y  +292.616, Z    +0.000, E1   +44.164, E3 +279968.234}
ENDSPLINE

SPLINE
SPL {X  -150.910, Y  +329.369, Z    +0.000, E1   +29.678, E3 +280040.630}
SPL {X  -156.829, Y  +350.854, Z    +0.000, E1   +20.141, E3 +280053.182}
SPL {X  -159.049, Y  +365.169, Z    +0.000, E1   +12.580, E3 +280057.926}
SPL {X  -159.776, Y  +374.231, Z    +0.000, E1    +7.281, E3 +280059.813}
SPL {X  -159.986, Y  +381.380, Z    +0.000, E1    +2.685, E3 +280060.659}
SPL {X  -159.990, Y  +385.261, Z    +0.000, E1    -0.259, E3 +280060.912}
SPL {X  -159.990, Y  +388.094, Z    +0.000, E1    -3.012, E3 +280061.104}
SPL {X  -159.990, Y  +390.622, Z    +0.000, E1    -5.876, E3 +280061.343}
SPL {X  -159.990, Y  +394.493, Z    +0.000, E1   -10.512, E3 +280061.866}
SPL {X  -159.990, Y  +401.377, Z    +0.000, E1   -19.398, E3 +280063.320}
SPL {X  -159.990, Y  +411.365, Z    +0.000, E1   -30.630, E3 +280066.529}
SPL {X  -159.990, Y  +450.467, Z    +0.000, E1   -50.183, E3 +280090.177}
SPL {X  -159.990, Y  +509.934, Z    +0.000, E1   -54.923, E3 +280152.796}
SPL {X  -159.990, Y  +516.848, Z    +0.000, E1   -54.930, E3 +280163.084}
SPL {X  -159.990, Y  +524.818, Z    +0.000, E1   -54.933, E3 +280174.956}
SPL {X  -159.990, Y  +532.100, Z    +0.000, E1   -54.924, E3 +280185.809}
SPL {X  -159.990, Y  +539.391, Z    +0.000, E1   -54.933, E3 +280196.661}
SPL {X  -159.990, Y  +546.283, Z    +0.000, E1   -54.924, E3 +280206.933}
SPL {X  -159.990, Y  +553.734, Z    +0.000, E1   -54.938, E3 +280218.020}
SPL {X  -159.990, Y  +564.956, Z    +0.000, E1   -54.973, E3 +280234.691}
SPL {X  -159.990, Y  +577.902, Z    +0.000, E1   -54.969, E3 +280253.981}
SPL {X  -159.990, Y  +588.063, Z    +0.000, E1   -54.931, E3 +280269.172}
SPL {X  -159.990, Y  +595.273, Z    +0.000, E1   -54.928, E3 +280279.895}
SPL {X  -159.990, Y  +602.326, Z    +0.000, E1   -54.932, E3 +280290.395}
SPL {X  -159.990, Y  +610.296, Z    +0.000, E1   -54.937, E3 +280302.265}
SPL {X  -159.990, Y  +618.534, Z    +0.000, E1   -54.942, E3 +280314.502}
SPL {X  -159.990, Y  +625.928, Z    +0.000, E1   -54.931, E3 +280325.527}
SPL {X  -159.990, Y  +633.423, Z    +0.000, E1   -54.943, E3 +280336.669}
SPL {X  -159.990, Y  +640.333, Z    +0.000, E1   -54.927, E3 +280346.983}
SPL {X  -159.990, Y  +648.272, Z    +0.000, E1   -54.961, E3 +280358.731}
SPL {X  -159.990, Y  +655.990, Z    +0.000, E1   -54.930, E3 +280370.278}
SPL {X  -159.990, Y  +665.734, Z    +0.000, E1   -54.984, E3 +280384.729}
SPL {X  -159.827, Y  +678.718, Z    +0.000, E1   -54.950, E3 +280404.258}
SPL {X  -159.222, Y  +687.156, Z    +0.000, E1   -54.792, E3 +280417.569}
SPL {X  -158.388, Y  +694.082, Z    +0.000, E1   -54.679, E3 +280428.706}
SPL {X  -157.277, Y  +700.838, Z    +0.000, E1   -54.465, E3 +280439.963}
SPL {X  -156.153, Y  +706.327, Z    +0.000, E1   -54.274, E3 +280449.299}
SPL {X  -154.917, Y  +711.470, Z    +0.000, E1   -54.052, E3 +280458.251}
SPL {X  -153.204, Y  +717.603, Z    +0.000, E1   -53.775, E3 +280469.097}
SPL {X  -151.355, Y  +723.351, Z    +0.000, E1   -53.415, E3 +280479.568}
SPL {X  -149.371, Y  +728.816, Z    +0.000, E1   -53.074, E3 +280489.659}
SPL {X  -147.376, Y  +733.767, Z    +0.000, E1   -52.671, E3 +280499.061}
SPL {X  -145.158, Y  +738.775, Z    +0.000, E1   -52.288, E3 +280508.612}
SPL {X  -142.385, Y  +744.461, Z    +0.000, E1   -51.729, E3 +280519.724}
SPL {X  -132.301, Y  +761.463, Z    +0.000, E1   -45.510, E3 +280597.463}
ENDSPLINE

SPLINE
SPL {X  -145.877, Y  +737.201, Z    +0.000, E1   -34.468, E3 +280680.574}
SPL {X  -152.550, Y  +719.721, Z    +0.000, E1   -27.728, E3 +280696.063}
SPL {X  -157.145, Y  +701.536, Z    +0.000, E1   -19.368, E3 +280705.517}
SPL {X  -159.035, Y  +688.952, Z    +0.000, E1   -12.676, E3 +280709.558}
SPL {X  -159.756, Y  +680.154, Z    +0.000, E1    -7.520, E3 +280711.285}
SPL {X  -159.986, Y  +672.560, Z    +0.000, E1    -2.636, E3 +280712.183}
SPL {X  -159.990, Y  +668.344, Z    +0.000, E1    +0.618, E3 +280712.449}
SPL {X  -159.990, Y  +664.070, Z    +0.000, E1    +5.025, E3 +280712.777}
SPL {X  -159.990, Y  +656.953, Z    +0.000, E1   +13.960, E3 +280713.844}
SPL {X  -159.990, Y  +644.589, Z    +0.000, E1   +29.011, E3 +280717.255}
SPL {X  -159.990, Y  +605.095, Z    +0.000, E1   +49.514, E3 +280742.346}
SPL {X  -159.990, Y  +543.998, Z    +0.000, E1   +54.483, E3 +280808.336}
SPL {X  -159.990, Y  +535.878, Z    +0.000, E1   +54.465, E3 +280820.671}
SPL {X  -159.990, Y  +529.394, Z    +0.000, E1   +54.464, E3 +280830.501}
SPL {X  -159.990, Y  +521.536, Z    +0.000, E1   +54.480, E3 +280842.382}
SPL {X  -159.990, Y  +514.089, Z    +0.000, E1   +54.461, E3 +280853.695}
SPL {X  -159.990, Y  +506.373, Z    +0.000, E1   +54.484, E3 +280865.331}
SPL {X  -159.990, Y  +497.571, Z    +0.000, E1   +54.478, E3 +280878.674}
SPL {X  -159.990, Y  +490.343, Z    +0.000, E1   +54.468, E3 +280889.639}
SPL {X  -159.990, Y  +483.191, Z    +0.000, E1   +54.478, E3 +280900.455}
SPL {X  -159.990, Y  +471.543, Z    +0.000, E1   +55.096, E3 +280914.083}
SPL {X  -159.990, Y  +443.253, Z    +0.000, E1   +59.297, E3 +280925.515}
SPL {X  -159.990, Y  +438.044, Z    +0.000, E1   +58.687, E3 +280936.370}
SPL {X  -159.990, Y  +431.936, Z    +0.000, E1   +57.955, E3 +280949.190}
SPL {X  -159.990, Y  +427.860, Z    +0.000, E1   +57.091, E3 +280960.253}
SPL {X  -159.990, Y  +424.653, Z    +0.000, E1   +55.901, E3 +280972.559}
SPL {X  -159.990, Y  +418.232, Z    +0.000, E1   +55.048, E3 +280987.352}
SPL {X  -159.990, Y  +410.722, Z    +0.000, E1   +54.900, E3 +280999.335}
SPL {X  -159.990, Y  +402.790, Z    +0.000, E1   +54.930, E3 +281011.110}
SPL {X  -159.990, Y  +391.119, Z    +0.000, E1   +54.948, E3 +281028.487}
SPL {X  -159.951, Y  +378.972, Z    +0.000, E1   +54.929, E3 +281046.666}
SPL {X  -159.499, Y  +369.977, Z    +0.000, E1   +54.827, E3 +281060.578}
SPL {X  -158.803, Y  +363.045, Z    +0.000, E1   +54.709, E3 +281071.647}
SPL {X  -157.966, Y  +357.131, Z    +0.000, E1   +54.559, E3 +281081.349}
SPL {X  -156.775, Y  +350.586, Z    +0.000, E1   +54.373, E3 +281092.323}
SPL {X  -155.027, Y  +342.959, Z    +0.000, E1   +54.074, E3 +281105.496}
SPL {X  -152.882, Y  +335.340, Z    +0.000, E1   +53.695, E3 +281119.039}
SPL {X  -151.019, Y  +329.680, Z    +0.000, E1   +53.334, E3 +281129.396}
SPL {X  -149.351, Y  +325.131, Z    +0.000, E1   +53.025, E3 +281137.840}
SPL {X  -147.860, Y  +321.391, Z    +0.000, E1   +52.740, E3 +281144.893}
SPL {X  -145.914, Y  +316.881, Z    +0.000, E1   +52.402, E3 +281153.462}
SPL {X  -142.795, Y  +310.344, Z    +0.000, E1   +51.829, E3 +281166.118}
SPL {X  -132.354, Y  +292.616, Z    +0.000, E1   +44.164, E3 +281264.530}
ENDSPLINE

SPLINE
SPL {X  -150.910, Y  +329.369, Z    +0.000, E1   +29.678, E3 +281336.926}
SPL {X  -156.396, Y  +348.778, Z    +0.000, E1   +21.134, E3 +281348.569}
SPL {X  -158.554, Y  +361.116, Z    +0.000, E1   +14.883, E3 +281353.023}
SPL {X  -159.881, Y  +376.607, Z    +0.000, E1    +5.865, E3 +281356.432}
SPL {X  -159.990, Y  +383.659, Z    +0.000, E1    +1.050, E3 +281357.113}
SPL {X  -159.990, Y  +387.327, Z    +0.000, E1    -2.137, E3 +281357.346}
SPL {X  -159.990, Y  +390.622, Z    +0.000, E1    -5.876, E3 +281357.639}
SPL {X  -159.990, Y  +394.493, Z    +0.000, E1   -10.512, E3 +281358.162}
SPL {X  -159.990, Y  +401.377, Z    +0.000, E1   -19.398, E3 +281359.616}
SPL {X  -159.990, Y  +411.365, Z    +0.000, E1   -30.630, E3 +281362.825}
SPL {X  -159.990, Y  +450.467, Z    +0.000, E1   -50.183, E3 +281386.474}
SPL {X  -159.990, Y  +509.934, Z    +0.000, E1   -54.923, E3 +281449.093}
SPL {X  -159.990, Y  +516.848, Z    +0.000, E1   -54.930, E3 +281459.381}
SPL {X  -159.990, Y  +524.818, Z    +0.000, E1   -54.933, E3 +281471.252}
SPL {X  -159.990, Y  +532.100, Z    +0.000, E1   -54.924, E3 +281482.106}
SPL {X  -159.990, Y  +539.391, Z    +0.000, E1   -54.933, E3 +281492.958}
SPL {X  -159.990, Y  +546.283, Z    +0.000, E1   -54.924, E3 +281503.229}
SPL {X  -159.990, Y  +553.734, Z    +0.000, E1   -54.938, E3 +281514.316}
SPL {X  -159.990, Y  +564.956, Z    +0.000, E1   -54.973, E3 +281530.987}
SPL {X  -159.990, Y  +577.902, Z    +0.000, E1   -54.969, E3 +281550.277}
SPL {X  -159.990, Y  +588.063, Z    +0.000, E1   -54.931, E3 +281565.468}
SPL {X  -159.990, Y  +595.273, Z    +0.000, E1   -54.928, E3 +281576.191}
SPL {X  -159.990, Y  +602.326, Z    +0.000, E1   -54.932, E3 +281586.692}
SPL {X  -159.990, Y  +610.296, Z    +0.000, E1   -54.937, E3 +281598.561}
SPL {X  -159.990, Y  +618.534, Z    +0.000, E1   -54.942, E3 +281610.798}
SPL {X  -159.990, Y  +628.178, Z    +0.000, E1   -54.959, E3 +281625.129}
SPL {X  -159.990, Y  +638.304, Z    +0.000, E1   -54.952, E3 +281640.218}
SPL {X  -159.990, Y  +648.272, Z    +0.000, E1   -54.961, E3 +281655.027}
SPL {X  -159.990, Y  +655.990, Z    +0.000, E1   -54.930, E3 +281666.575}
SPL {X  -159.990, Y  +665.734, Z    +0.000, E1   -54.984, E3 +281681.026}
SPL {X  -159.827, Y  +678.718, Z    +0.000, E1   -54.950, E3 +281700.554}
SPL {X  -159.222, Y  +687.156, Z    +0.000, E1   -54.792, E3 +281713.865}
SPL {X  -158.388, Y  +694.082, Z    +0.000, E1   -54.679, E3 +281725.003}
SPL {X  -157.277, Y  +700.838, Z    +0.000, E1   -54.465, E3 +281736.260}
SPL {X  -156.153, Y  +706.327, Z    +0.000, E1   -54.274, E3 +281745.596}
SPL {X  -154.917, Y  +711.470, Z    +0.000, E1   -54.052, E3 +281754.547}
SPL {X  -153.204, Y  +717.603, Z    +0.000, E1   -53.775, E3 +281765.393}
SPL {X  -151.355, Y  +723.351, Z    +0.000, E1   -53.415, E3 +281775.864}
SPL {X  -149.371, Y  +728.816, Z    +0.000, E1   -53.074, E3 +281785.955}
SPL {X  -147.376, Y  +733.767, Z    +0.000, E1   -52.671, E3 +281795.357}
SPL {X  -145.158, Y  +738.775, Z    +0.000, E1   -52.288, E3 +281804.908}
SPL {X  -142.385, Y  +744.461, Z    +0.000, E1   -51.729, E3 +281816.020}
SPL {X  -132.301, Y  +761.463, Z    +0.000, E1   -45.510, E3 +281893.759}
ENDSPLINE

SPLINE
SPL {X  -145.877, Y  +737.201, Z    +0.000, E1   -34.468, E3 +281976.870}
SPL {X  -152.550, Y  +719.721, Z    +0.000, E1   -27.728, E3 +281992.359}
SPL {X  -157.145, Y  +701.536, Z    +0.000, E1   -19.368, E3 +282001.814}
SPL {X  -159.035, Y  +688.952, Z    +0.000, E1   -12.676, E3 +282005.855}
SPL {X  -159.756, Y  +680.154, Z    +0.000, E1    -7.520, E3 +282007.581}
SPL {X  -159.986, Y  +672.560, Z    +0.000, E1    -2.636, E3 +282008.479}
SPL {X  -159.990, Y  +668.344, Z    +0.000, E1    +0.618, E3 +282008.745}
SPL {X  -159.990, Y  +664.070, Z    +0.000, E1    +5.025, E3 +282009.074}
SPL {X  -159.990, Y  +656.953, Z    +0.000, E1   +13.960, E3 +282010.140}
SPL {X  -159.990, Y  +644.589, Z    +0.000, E1   +29.011, E3 +282013.552}
SPL {X  -159.990, Y  +605.095, Z    +0.000, E1   +49.514, E3 +282038.643}
SPL {X  -159.990, Y  +546.155, Z    +0.000, E1   +54.461, E3 +282101.401}
SPL {X  -159.990, Y  +537.700, Z    +0.000, E1   +54.492, E3 +282114.165}
SPL {X  -159.990, Y  +529.394, Z    +0.000, E1   +54.464, E3 +282126.797}
SPL {X  -159.990, Y  +521.536, Z    +0.000, E1   +54.480, E3 +282138.678}
SPL {X  -159.990, Y  +514.089, Z    +0.000, E1   +54.461, E3 +282149.991}
SPL {X  -159.990, Y  +506.373, Z    +0.000, E1   +54.484, E3 +282161.627}
SPL {X  -159.990, Y  +497.571, Z    +0.000, E1   +54.478, E3 +282174.970}
SPL {X  -159.990, Y  +490.343, Z    +0.000, E1   +54.468, E3 +282185.935}
SPL {X  -159.990, Y  +483.191, Z    +0.000, E1   +54.478, E3 +282196.751}
SPL {X  -159.990, Y  +475.502, Z    +0.000, E1   +54.476, E3 +282208.401}
SPL {X  -159.990, Y  +448.520, Z    +0.000, E1   +58.543, E3 +282220.030}
SPL {X  -159.990, Y  +438.044, Z    +0.000, E1   +58.687, E3 +282232.667}
SPL {X  -159.990, Y  +431.936, Z    +0.000, E1   +57.955, E3 +282245.486}
SPL {X  -159.990, Y  +427.860, Z    +0.000, E1   +57.091, E3 +282256.550}
SPL {X  -159.990, Y  +424.653, Z    +0.000, E1   +55.901, E3 +282268.855}
SPL {X  -159.990, Y  +418.232, Z    +0.000, E1   +55.048, E3 +282283.648}
SPL {X  -159.990, Y  +410.722, Z    +0.000, E1   +54.900, E3 +282295.631}
SPL {X  -159.990, Y  +402.790, Z    +0.000, E1   +54.930, E3 +282307.406}
SPL {X  -159.990, Y  +392.953, Z    +0.000, E1   +54.918, E3 +282322.100}
SPL {X  -159.990, Y  +383.354, Z    +0.000, E1   +54.920, E3 +282336.410}
SPL {X  -159.860, Y  +376.053, Z    +0.000, E1   +54.872, E3 +282347.470}
SPL {X  -159.499, Y  +369.977, Z    +0.000, E1   +54.827, E3 +282356.874}
SPL {X  -158.803, Y  +363.045, Z    +0.000, E1   +54.709, E3 +282367.943}
SPL {X  -157.732, Y  +355.717, Z    +0.000, E1   +54.540, E3 +282379.965}
SPL {X  -156.235, Y  +348.039, Z    +0.000, E1   +54.281, E3 +282392.977}
SPL {X  -154.716, Y  +341.761, Z    +0.000, E1   +53.995, E3 +282403.934}
SPL {X  -152.882, Y  +335.340, Z    +0.000, E1   +53.695, E3 +282415.335}
SPL {X  -151.019, Y  +329.680, Z    +0.000, E1   +53.334, E3 +282425.692}
SPL {X  -149.351, Y  +325.131, Z    +0.000, E1   +53.025, E3 +282434.136}
SPL {X  -147.860, Y  +321.391, Z    +0.000, E1   +52.740, E3 +282441.189}
SPL {X  -145.914, Y  +316.881, Z    +0.000, E1   +52.402, E3 +282449.759}
SPL {X  -142.795, Y  +310.344, Z    +0.000, E1   +51.829, E3 +282462.414}
SPL {X  -132.354, Y  +292.616, Z    +0.000, E1   +44.164, E3 +282560.827}
ENDSPLINE

SPLINE
SPL {X  -150.910, Y  +329.369, Z    +0.000, E1   +29.678, E3 +282633.222}
SPL {X  -156.829, Y  +350.854, Z    +0.000, E1   +20.141, E3 +282645.775}
SPL {X  -159.049, Y  +365.169, Z    +0.000, E1   +12.580, E3 +282650.519}
SPL {X  -159.776, Y  +374.231, Z    +0.000, E1    +7.281, E3 +282652.405}
SPL {X  -159.986, Y  +381.380, Z    +0.000, E1    +2.685, E3 +282653.251}
SPL {X  -159.990, Y  +384.493, Z    +0.000, E1    +0.324, E3 +282653.459}
SPL {X  -159.990, Y  +387.327, Z    +0.000, E1    -2.137, E3 +282653.642}
SPL {X  -159.990, Y  +392.053, Z    +0.000, E1    -7.477, E3 +282654.107}
SPL {X  -159.990, Y  +396.158, Z    +0.000, E1   -12.775, E3 +282654.732}
SPL {X  -159.990, Y  +401.377, Z    +0.000, E1   -19.398, E3 +282655.913}
SPL {X  -159.990, Y  +411.365, Z    +0.000, E1   -30.630, E3 +282659.121}
SPL {X  -159.990, Y  +450.467, Z    +0.000, E1   -50.183, E3 +282682.770}
SPL {X  -159.990, Y  +509.934, Z    +0.000, E1   -54.923, E3 +282745.389}
SPL {X  -159.990, Y  +516.848, Z    +0.000, E1   -54.930, E3 +282755.677}
SPL {X  -159.990, Y  +524.818, Z    +0.000, E1   -54.933, E3 +282767.549}
SPL {X  -159.990, Y  +532.100, Z    +0.000, E1   -54.924, E3 +282778.402}
SPL {X  -159.990, Y  +539.391, Z    +0.000, E1   -54.933, E3 +282789.254}
SPL {X  -159.990, Y  +546.283, Z    +0.000, E1   -54.924, E3 +282799.525}
SPL {X  -159.990, Y  +553.734, Z    +0.000, E1   -54.938, E3 +282810.612}
SPL {X  -159.990, Y  +560.983, Z    +0.000, E1   -54.918, E3 +282821.450}
SPL {X  -159.990, Y  +567.462, Z    +0.000, E1   -54.929, E3 +282831.085}
SPL {X  -159.990, Y  +575.140, Z    +0.000, E1   -54.928, E3 +282842.517}
SPL {X  -159.990, Y  +581.046, Z    +0.000, E1   -54.920, E3 +282851.329}
SPL {X  -159.990, Y  +588.063, Z    +0.000, E1   -54.931, E3 +282861.764}
SPL {X  -159.990, Y  +595.273, Z    +0.000, E1   -54.928, E3 +282872.488}
SPL {X  -159.990, Y  +602.326, Z    +0.000, E1   -54.932, E3 +282882.988}
SPL {X  -159.990, Y  +610.296, Z    +0.000, E1   -54.937, E3 +282894.857}
SPL {X  -159.990, Y  +618.534, Z    +0.000, E1   -54.942, E3 +282907.094}
SPL {X  -159.990, Y  +625.928, Z    +0.000, E1   -54.931, E3 +282918.120}
SPL {X  -159.990, Y  +633.423, Z    +0.000, E1   -54.943, E3 +282929.262}
SPL {X  -159.990, Y  +643.352, Z    +0.000, E1   -54.966, E3 +282943.997}
SPL {X  -159.990, Y  +650.756, Z    +0.000, E1   -54.931, E3 +282955.064}
SPL {X  -159.990, Y  +658.525, Z    +0.000, E1   -54.959, E3 +282966.600}
SPL {X  -159.990, Y  +667.903, Z    +0.000, E1   -54.941, E3 +282980.631}
SPL {X  -159.953, Y  +674.920, Z    +0.000, E1   -54.918, E3 +282991.134}
SPL {X  -159.714, Y  +680.893, Z    +0.000, E1   -54.890, E3 +283000.274}
SPL {X  -159.222, Y  +687.156, Z    +0.000, E1   -54.792, E3 +283010.161}
SPL {X  -158.388, Y  +694.082, Z    +0.000, E1   -54.679, E3 +283021.299}
SPL {X  -157.277, Y  +700.838, Z    +0.000, E1   -54.465, E3 +283032.556}
SPL {X  -156.153, Y  +706.327, Z    +0.000, E1   -54.274, E3 +283041.892}
SPL {X  -154.917, Y  +711.470, Z    +0.000, E1   -54.052, E3 +283050.843}
SPL {X  -153.204, Y  +717.603, Z    +0.000, E1   -53.775, E3 +283061.689}
SPL {X  -151.355, Y  +723.351, Z    +0.000, E1   -53.415, E3 +283072.161}
SPL {X  -149.371, Y  +728.816, Z    +0.000, E1   -53.074, E3 +283082.251}
SPL {X  -146.631, Y  +735.501, Z    +0.000, E1   -52.568, E3 +283094.912}
SPL {X  -144.428, Y  +740.329, Z    +0.000, E1   -52.109, E3 +283104.266}
SPL {X  -142.385, Y  +744.461, Z    +0.000, E1   -51.729, E3 +283112.317}
SPL {X  -132.301, Y  +761.463, Z    +0.000, E1   -45.510, E3 +283190.055}
ENDSPLINE

SPLINE
SPL {X  -145.877, Y  +737.201, Z    +0.000, E1   -34.468, E3 +283273.166}
SPL {X  -152.550, Y  +719.721, Z    +0.000, E1   -27.728, E3 +283288.655}
SPL {X  -157.145, Y  +701.536, Z    +0.000, E1   -19.368, E3 +283298.110}
SPL {X  -159.035, Y  +688.952, Z    +0.000, E1   -12.676, E3 +283302.151}
SPL {X  -159.756, Y  +680.154, Z    +0.000, E1    -7.520, E3 +283303.877}
SPL {X  -159.986, Y  +672.560, Z    +0.000, E1    -2.636, E3 +283304.776}
SPL {X  -159.990, Y  +668.344, Z    +0.000, E1    +0.618, E3 +283305.042}
SPL {X  -159.990, Y  +664.070, Z    +0.000, E1    +5.025, E3 +283305.370}
SPL {X  -159.990, Y  +656.953, Z    +0.000, E1   +13.960, E3 +283306.437}
SPL {X  -159.990, Y  +644.589, Z    +0.000, E1   +29.011, E3 +283309.848}
SPL {X  -159.990, Y  +605.095, Z    +0.000, E1   +49.514, E3 +283334.939}
SPL {X  -159.990, Y  +543.998, Z    +0.000, E1   +54.483, E3 +283400.929}
SPL {X  -159.990, Y  +535.878, Z    +0.000, E1   +54.465, E3 +283413.264}
SPL {X  -159.990, Y  +529.394, Z    +0.000, E1   +54.464, E3 +283423.093}
SPL {X  -159.990, Y  +521.536, Z    +0.000, E1   +54.480, E3 +283434.975}
SPL {X  -159.990, Y  +512.119, Z    +0.000, E1   +54.487, E3 +283449.221}
SPL {X  -159.990, Y  +504.581, Z    +0.000, E1   +54.460, E3 +283460.680}
SPL {X  -159.990, Y  +497.571, Z    +0.000, E1   +54.478, E3 +283471.267}
SPL {X  -159.990, Y  +490.343, Z    +0.000, E1   +54.468, E3 +283482.232}
SPL {X  -159.990, Y  +483.191, Z    +0.000, E1   +54.478, E3 +283493.048}
SPL {X  -159.990, Y  +475.502, Z    +0.000, E1   +54.476, E3 +283504.697}
SPL {X  -159.990, Y  +448.520, Z    +0.000, E1   +58.543, E3 +283516.326}
SPL {X  -159.990, Y  +438.044, Z    +0.000, E1   +58.687, E3 +283528.963}
SPL {X  -159.990, Y  +431.936, Z    +0.000, E1   +57.955, E3 +283541.782}
SPL {X  -159.990, Y  +427.293, Z    +0.000, E1   +56.830, E3 +283555.488}
SPL {X  -159.990, Y  +423.841, Z    +0.000, E1   +55.679, E3 +283567.590}
SPL {X  -159.990, Y  +418.232, Z    +0.000, E1   +55.048, E3 +283579.944}
SPL {X  -159.990, Y  +410.722, Z    +0.000, E1   +54.900, E3 +283591.927}
SPL {X  -159.990, Y  +402.790, Z    +0.000, E1   +54.930, E3 +283603.702}
SPL {X  -159.990, Y  +392.953, Z    +0.000, E1   +54.918, E3 +283618.396}
SPL {X  -159.990, Y  +383.354, Z    +0.000, E1   +54.920, E3 +283632.706}
SPL {X  -159.660, Y  +372.225, Z    +0.000, E1   +54.896, E3 +283649.587}
SPL {X  -158.803, Y  +363.045, Z    +0.000, E1   +54.709, E3 +283664.239}
SPL {X  -157.732, Y  +355.717, Z    +0.000, E1   +54.540, E3 +283676.262}
SPL {X  -156.235, Y  +348.039, Z    +0.000, E1   +54.281, E3 +283689.273}
SPL {X  -154.716, Y  +341.761, Z    +0.000, E1   +53.995, E3 +283700.230}
SPL {X  -152.882, Y  +335.340, Z    +0.000, E1   +53.695, E3 +283711.632}
SPL {X  -151.019, Y  +329.680, Z    +0.000, E1   +53.334, E3 +283721.989}
SPL {X  -148.682, Y  +323.421, Z    +0.000, E1   +52.939, E3 +283733.591}
SPL {X  -145.914, Y  +316.881, Z    +0.000, E1   +52.402, E3 +283746.055}
SPL {X  -142.795, Y  +310.344, Z    +0.000, E1   +51.829, E3 +283758.711}
SPL {X  -132.354, Y  +292.616, Z    +0.000, E1   +44.164, E3 +283857.123}
ENDSPLINE

SPLINE
SPL {X  -150.910, Y  +329.369, Z    +0.000, E1   +29.678, E3 +283929.518}
SPL {X  -156.396, Y  +348.778, Z    +0.000, E1   +21.134, E3 +283941.162}
SPL {X  -158.554, Y  +361.116, Z    +0.000, E1   +14.883, E3 +283945.616}
SPL {X  -159.881, Y  +376.607, Z    +0.000, E1    +5.865, E3 +283949.025}
SPL {X  -159.990, Y  +383.659, Z    +0.000, E1    +1.050, E3 +283949.705}
SPL {X  -159.990, Y  +387.327, Z    +0.000, E1    -2.137, E3 +283949.938}
SPL {X  -159.990, Y  +390.622, Z    +0.000, E1    -5.876, E3 +283950.231}
SPL {X  -159.990, Y  +394.493, Z    +0.000, E1   -10.512, E3 +283950.754}
SPL {X  -159.990, Y  +401.377, Z    +0.000, E1   -19.398, E3 +283952.209}
SPL {X  -159.990, Y  +411.365, Z    +0.000, E1   -30.630, E3 +283955.417}
SPL {X  -159.990, Y  +450.467, Z    +0.000, E1   -50.183, E3 +283979.066}
SPL {X  -159.990, Y  +509.934, Z    +0.000, E1   -54.923, E3 +284041.685}
SPL {X  -159.990, Y  +516.848, Z    +0.000, E1   -54.930, E3 +284051.973}
SPL {X  -159.990, Y  +524.818, Z    +0.000, E1   -54.933, E3 +284063.845}
SPL {X  -159.990, Y  +532.100, Z    +0.000, E1   -54.924, E3 +284074.698}
SPL {X  -159.990, Y  +539.391, Z    +0.000, E1   -54.933, E3 +284085.550}
SPL {X  -159.990, Y  +546.283, Z    +0.000, E1   -54.924, E3 +284095.822}
SPL {X  -159.990, Y  +553.734, Z    +0.000, E1   -54.938, E3 +284106.908}
SPL {X  -159.990, Y  +564.956, Z    +0.000, E1   -54.973, E3 +284123.580}
SPL {X  -159.990, Y  +577.902, Z    +0.000, E1   -54.969, E3 +284142.870}
SPL {X  -159.990, Y  +588.063, Z    +0.000, E1   -54.931, E3 +284158.060}
SPL {X  -159.990, Y  +595.273, Z    +0.000, E1   -54.928, E3 +284168.784}
SPL {X  -159.990, Y  +602.326, Z    +0.000, E1   -54.932, E3 +284179.284}
SPL {X  -159.990, Y  +610.296, Z    +0.000, E1   -54.937, E3 +284191.154}
SPL {X  -159.990, Y  +618.534, Z    +0.000, E1   -54.942, E3 +284203.391}
SPL {X  -159.990, Y  +625.928, Z    +0.000, E1   -54.931, E3 +284214.416}
SPL {X  -159.990, Y  +633.423, Z    +0.000, E1   -54.943, E3 +284225.558}
SPL {X  -159.990, Y  +640.333, Z    +0.000, E1   -54.927, E3 +284235.872}
SPL {X  -159.990, Y  +648.272, Z    +0.000, E1   -54.961, E3 +284247.620}
SPL {X  -159.990, Y  +655.990, Z    +0.000, E1   -54.930, E3 +284259.167}
SPL {X  -159.990, Y  +665.734, Z    +0.000, E1   -54.984, E3 +284273.618}
SPL {X  -159.827, Y  +678.718, Z    +0.000, E1   -54.950, E3 +284293.147}
SPL {X  -159.222, Y  +687.156, Z    +0.000, E1   -54.792, E3 +284306.457}
SPL {X  -158.388, Y  +694.082, Z    +0.000, E1   -54.679, E3 +284317.595}
SPL {X  -157.277, Y  +700.838, Z    +0.000, E1   -54.465, E3 +284328.852}
SPL {X  -156.153, Y  +706.327, Z    +0.000, E1   -54.274, E3 +284338.188}
SPL {X  -154.917, Y  +711.470, Z    +0.000, E1   -54.052, E3 +284347.140}
SPL {X  -153.204, Y  +717.603, Z    +0.000, E1   -53.775, E3 +284357.986}
SPL {X  -151.355, Y  +723.351, Z    +0.000, E1   -53.415, E3 +284368.457}
SPL {X  -149.371, Y  +728.816, Z    +0.000, E1   -53.074, E3 +284378.548}
SPL {X  -146.631, Y  +735.501, Z    +0.000, E1   -52.568, E3 +284391.208}
SPL {X  -144.428, Y  +740.329, Z    +0.000, E1   -52.109, E3 +284400.562}
SPL {X  -142.385, Y  +744.461, Z    +0.000, E1   -51.729, E3 +284408.613}
SPL {X  -132.301, Y  +761.463, Z    +0.000, E1   -45.510, E3 +284486.352}
ENDSPLINE

SPLINE
SPL {X  -145.877, Y  +737.201, Z    +0.000, E1   -34.468, E3 +284569.463}
SPL {X  -152.550, Y  +719.721, Z    +0.000, E1   -27.728, E3 +284584.952}
SPL {X  -157.145, Y  +701.536, Z    +0.000, E1   -19.368, E3 +284594.406}
SPL {X  -159.035, Y  +688.952, Z    +0.000, E1   -12.676, E3 +284598.447}
SPL {X  -159.873, Y  +677.622, Z    +0.000, E1    -6.008, E3 +284600.519}
SPL {X  -159.990, Y  +671.638, Z    +0.000, E1    -1.925, E3 +284601.146}
SPL {X  -159.990, Y  +668.344, Z    +0.000, E1    +0.618, E3 +284601.338}
SPL {X  -159.990, Y  +665.430, Z    +0.000, E1    +3.630, E3 +284601.533}
SPL {X  -159.990, Y  +661.750, Z    +0.000, E1    +7.880, E3 +284601.924}
SPL {X  -159.990, Y  +655.696, Z    +0.000, E1   +15.733, E3 +284602.976}
SPL {X  -159.990, Y  +644.589, Z    +0.000, E1   +29.011, E3 +284606.144}
SPL {X  -159.990, Y  +605.095, Z    +0.000, E1   +49.514, E3 +284631.235}
SPL {X  -159.990, Y  +543.998, Z    +0.000, E1   +54.483, E3 +284697.225}
SPL {X  -159.990, Y  +535.878, Z    +0.000, E1   +54.465, E3 +284709.560}
SPL {X  -159.990, Y  +529.394, Z    +0.000, E1   +54.464, E3 +284719.389}
SPL {X  -159.990, Y  +521.536, Z    +0.000, E1   +54.480, E3 +284731.271}
SPL {X  -159.990, Y  +512.119, Z    +0.000, E1   +54.487, E3 +284745.517}
SPL {X  -159.990, Y  +504.581, Z    +0.000, E1   +54.460, E3 +284756.976}
SPL {X  -159.990, Y  +497.571, Z    +0.000, E1   +54.478, E3 +284767.563}
SPL {X  -159.990, Y  +490.343, Z    +0.000, E1   +54.468, E3 +284778.528}
SPL {X  -159.990, Y  +483.191, Z    +0.000, E1   +54.478, E3 +284789.344}
SPL {X  -159.990, Y  +475.502, Z    +0.000, E1   +54.476, E3 +284800.993}
SPL {X  -159.990, Y  +448.520, Z    +0.000, E1   +58.543, E3 +284812.622}
SPL {X  -159.990, Y  +438.044, Z    +0.000, E1   +58.687, E3 +284825.259}
SPL {X  -159.990, Y  +431.936, Z    +0.000, E1   +57.955, E3 +284838.079}
SPL {X  -159.990, Y  +427.293, Z    +0.000, E1   +56.830, E3 +284851.785}
SPL {X  -159.990, Y  +423.841, Z    +0.000, E1   +55.679, E3 +284863.887}
SPL {X  -159.990, Y  +419.589, Z    +0.000, E1   +55.096, E3 +284873.811}
SPL {X  -159.990, Y  +412.636, Z    +0.000, E1   +54.925, E3 +284885.323}
SPL {X  -159.990, Y  +405.235, Z    +0.000, E1   +54.902, E3 +284896.393}
SPL {X  -159.990, Y  +400.284, Z    +0.000, E1   +54.897, E3 +284903.788}
SPL {X  -159.990, Y  +392.953, Z    +0.000, E1   +54.918, E3 +284914.692}
SPL {X  -159.990, Y  +383.354, Z    +0.000, E1   +54.920, E3 +284929.002}
SPL {X  -159.769, Y  +374.091, Z    +0.000, E1   +54.882, E3 +284943.035}
SPL {X  -158.996, Y  +364.689, Z    +0.000, E1   +54.773, E3 +284957.831}
SPL {X  -157.966, Y  +357.131, Z    +0.000, E1   +54.559, E3 +284970.238}
SPL {X  -156.775, Y  +350.586, Z    +0.000, E1   +54.373, E3 +284981.212}
SPL {X  -155.027, Y  +342.959, Z    +0.000, E1   +54.074, E3 +284994.385}
SPL {X  -152.882, Y  +335.340, Z    +0.000, E1   +53.695, E3 +285007.928}
SPL {X  -151.019, Y  +329.680, Z    +0.000, E1   +53.334, E3 +285018.285}
SPL {X  -149.351, Y  +325.131, Z    +0.000, E1   +53.025, E3 +285026.729}
SPL {X  -147.860, Y  +321.391, Z    +0.000, E1   +52.740, E3 +285033.781}
SPL {X  -145.914, Y  +316.881, Z    +0.000, E1   +52.402, E3 +285042.351}
SPL {X  -142.795, Y  +310.344, Z    +0.000, E1   +51.829, E3 +285055.007}
SPL {X  -132.354, Y  +292.616, Z    +0.000, E1   +44.164, E3 +285153.419}
ENDSPLINE

SPLINE
SPL {X  -150.910, Y  +329.369, Z    +0.000, E1   +29.678, E3 +285225.815}
SPL {X  -156.396, Y  +348.778, Z    +0.000, E1   +21.134, E3 +285237.458}
SPL {X  -158.554, Y  +361.116, Z    +0.000, E1   +14.883, E3 +285241.912}
SPL {X  -159.881, Y  +376.607, Z    +0.000, E1    +5.865, E3 +285245.321}
SPL {X  -159.990, Y  +383.659, Z    +0.000, E1    +1.050, E3 +285246.002}
SPL {X  -159.990, Y  +387.327, Z    +0.000, E1    -2.137, E3 +285246.234}
SPL {X  -159.990, Y  +390.622, Z    +0.000, E1    -5.876, E3 +285246.528}
SPL {X  -159.990, Y  +394.493, Z    +0.000, E1   -10.512, E3 +285247.051}
SPL {X  -159.990, Y  +401.377, Z    +0.000, E1   -19.398, E3 +285248.505}
SPL {X  -159.990, Y  +411.365, Z    +0.000, E1   -30.630, E3 +285251.714}
SPL {X  -159.990, Y  +450.467, Z    +0.000, E1   -50.183, E3 +285275.363}
SPL {X  -159.990, Y  +509.934, Z    +0.000, E1   -54.923, E3 +285337.981}
SPL {X  -159.990, Y  +516.848, Z    +0.000, E1   -54.930, E3 +285348.269}
SPL {X  -159.990, Y  +524.818, Z    +0.000, E1   -54.933, E3 +285360.141}
SPL {X  -159.990, Y  +532.100, Z    +0.000, E1   -54.924, E3 +285370.994}
SPL {X  -159.990, Y  +539.391, Z    +0.000, E1   -54.933, E3 +285381.846}
SPL {X  -159.990, Y  +546.283, Z    +0.000, E1   -54.924, E3 +285392.118}
SPL {X  -159.990, Y  +553.734, Z    +0.000, E1   -54.938, E3 +285403.205}
SPL {X  -159.990, Y  +564.956, Z    +0.000, E1   -54.973, E3 +285419.876}
SPL {X  -159.990, Y  +577.902, Z    +0.000, E1   -54.969, E3 +285439.166}
SPL {X  -159.990, Y  +588.063, Z    +0.000, E1   -54.931, E3 +285454.357}
SPL {X  -159.990, Y  +595.273, Z    +0.000, E1   -54.928, E3 +285465.080}
SPL {X  -159.990, Y  +602.326, Z    +0.000, E1   -54.932, E3 +285475.581}
SPL {X  -159.990, Y  +610.296, Z    +0.000, E1   -54.937, E3 +285487.450}
SPL {X  -159.990, Y  +618.534, Z    +0.000, E1   -54.942, E3 +285499.687}
SPL {X  -159.990, Y  +628.178, Z    +0.000, E1   -54.959, E3 +285514.018}
SPL {X  -159.990, Y  +638.304, Z    +0.000, E1   -54.952, E3 +285529.107}
SPL {X  -159.990, Y  +648.272, Z    +0.000, E1   -54.961, E3 +285543.916}
SPL {X  -159.990, Y  +655.990, Z    +0.000, E1   -54.930, E3 +285555.464}
SPL {X  -159.990, Y  +665.734, Z    +0.000, E1   -54.984, E3 +285569.915}
SPL {X  -159.827, Y  +678.718, Z    +0.000, E1   -54.950, E3 +285589.443}
SPL {X  -159.222, Y  +687.156, Z    +0.000, E1   -54.792, E3 +285602.754}
SPL {X  -158.388, Y  +694.082, Z    +0.000, E1   -54.679, E3 +285613.891}
SPL {X  -157.277, Y  +700.838, Z    +0.000, E1   -54.465, E3 +285625.149}
SPL {X  -156.153, Y  +706.327, Z    +0.000, E1   -54.274, E3 +285634.485}
SPL {X  -154.917, Y  +711.470, Z    +0.000, E1   -54.052, E3 +285643.436}
SPL {X  -153.204, Y  +717.603, Z    +0.000, E1   -53.775, E3 +285654.282}
SPL {X  -151.355, Y  +723.351, Z    +0.000, E1   -53.415, E3 +285664.753}
SPL {X  -149.371, Y  +728.816, Z    +0.000, E1   -53.074, E3 +285674.844}
SPL {X  -147.376, Y  +733.767, Z    +0.000, E1   -52.671, E3 +285684.246}
SPL {X  -145.158, Y  +738.775, Z    +0.000, E1   -52.288, E3 +285693.797}
SPL {X  -142.385, Y  +744.461, Z    +0.000, E1   -51.729, E3 +285704.909}
SPL {X  -132.301, Y  +761.463, Z    +0.000, E1   -45.510, E3 +285782.648}
ENDSPLINE

SPLINE
SPL {X  -145.877, Y  +737.201, Z    +0.000, E1   -34.468, E3 +285865.759}
SPL {X  -152.550, Y  +719.721, Z    +0.000, E1   -27.728, E3 +285881.248}
SPL {X  -157.145, Y  +701.536, Z    +0.000, E1   -19.368, E3 +285890.703}
SPL {X  -159.035, Y  +688.952, Z    +0.000, E1   -12.676, E3 +285894.744}
SPL {X  -159.756, Y  +680.154, Z    +0.000, E1    -7.520, E3 +285896.470}
SPL {X  -159.986, Y  +672.560, Z    +0.000, E1    -2.636, E3 +285897.368}
SPL {X  -159.990, Y  +668.344, Z    +0.000, E1    +0.618, E3 +285897.634}
SPL {X  -159.990, Y  +664.070, Z    +0.000, E1    +5.025, E3 +285897.963}
SPL {X  -159.990, Y  +656.953, Z    +0.000, E1   +13.960, E3 +285899.029}
SPL {X  -159.990, Y  +644.589, Z    +0.000, E1   +29.011, E3 +285902.441}
SPL {X  -159.990, Y  +605.095, Z    +0.000, E1   +49.514, E3 +285927.532}
SPL {X  -159.990, Y  +546.155, Z    +0.000, E1   +54.461, E3 +285990.290}
SPL {X  -159.990, Y  +537.700, Z    +0.000, E1   +54.492, E3 +286003.054}
SPL {X  -159.990, Y  +529.394, Z    +0.000, E1   +54.464, E3 +286015.686}
SPL {X  -159.990, Y  +521.536, Z    +0.000, E1   +54.480, E3 +286027.567}
SPL {X  -159.990, Y  +514.089, Z    +0.000, E1   +54.461, E3 +286038.880}
SPL {X  -159.990, Y  +506.373, Z    +0.000, E1   +54.484, E3 +286050.516}
SPL {X  -159.990, Y  +497.571, Z    +0.000, E1   +54.478, E3 +286063.859}
SPL {X  -159.990, Y  +490.343, Z    +0.000, E1   +54.468, E3 +286074.824}
SPL {X  -159.990, Y  +483.191, Z    +0.000, E1   +54.478, E3 +286085.640}
SPL {X  -159.990, Y  +475.502, Z    +0.000, E1   +54.476, E3 +286097.290}
SPL {X  -159.990, Y  +448.520, Z    +0.000, E1   +58.543, E3 +286108.919}
SPL {X  -159.990, Y  +438.044, Z    +0.000, E1   +58.687, E3 +286121.555}
SPL {X  -159.990, Y  +431.936, Z    +0.000, E1   +57.955, E3 +286134.375}
SPL {X  -159.990, Y  +427.860, Z    +0.000, E1   +57.091, E3 +286145.439}
SPL {X  -159.990, Y  +424.653, Z    +0.000, E1   +55.901, E3 +286157.744}
SPL {X  -159.990, Y  +418.232, Z    +0.000, E1   +55.048, E3 +286172.537}
SPL {X  -159.990, Y  +410.722, Z    +0.000, E1   +54.900, E3 +286184.520}
SPL {X  -159.990, Y  +402.790, Z    +0.000, E1   +54.930, E3 +286196.295}
SPL {X  -159.990, Y  +392.953, Z    +0.000, E1   +54.918, E3 +286210.989}
SPL {X  -159.990, Y  +383.354, Z    +0.000, E1   +54.920, E3 +286225.299}
SPL {X  -159.860, Y  +376.053, Z    +0.000, E1   +54.872, E3 +286236.358}
SPL {X  -159.499, Y  +369.977, Z    +0.000, E1   +54.827, E3 +286245.763}
SPL {X  -158.803, Y  +363.045, Z    +0.000, E1   +54.709, E3 +286256.832}
SPL {X  -157.732, Y  +355.717, Z    +0.000, E1   +54.540, E3 +286268.854}
SPL {X  -156.235, Y  +348.039, Z    +0.000, E1   +54.281, E3 +286281.866}
SPL {X  -154.716, Y  +341.761, Z    +0.000, E1   +53.995, E3 +286292.823}
SPL {X  -152.882, Y  +335.340, Z    +0.000, E1   +53.695, E3 +286304.224}
SPL {X  -151.019, Y  +329.680, Z    +0.000, E1   +53.334, E3 +286314.581}
SPL {X  -149.351, Y  +325.131, Z    +0.000, E1   +53.025, E3 +286323.025}
SPL {X  -147.860, Y  +321.391, Z    +0.000, E1   +52.740, E3 +286330.078}
SPL {X  -145.914, Y  +316.881, Z    +0.000, E1   +52.402, E3 +286338.648}
SPL {X  -142.795, Y  +310.344, Z    +0.000, E1   +51.829, E3 +286351.303}
SPL {X  -132.354, Y  +292.616, Z    +0.000, E1   +44.164, E3 +286449.716}
ENDSPLINE

SPLINE
SPL {X  -150.910, Y  +329.369, Z    +0.000, E1   +29.678, E3 +286522.111}
SPL {X  -156.829, Y  +350.854, Z    +0.000, E1   +20.141, E3 +286534.664}
SPL {X  -159.049, Y  +365.169, Z    +0.000, E1   +12.580, E3 +286539.408}
SPL {X  -159.776, Y  +374.231, Z    +0.000, E1    +7.281, E3 +286541.294}
SPL {X  -159.986, Y  +381.380, Z    +0.000, E1    +2.685, E3 +286542.140}
SPL {X  -159.990, Y  +384.493, Z    +0.000, E1    +0.324, E3 +286542.348}
SPL {X  -159.990, Y  +387.327, Z    +0.000, E1    -2.137, E3 +286542.531}
SPL {X  -159.990, Y  +392.053, Z    +0.000, E1    -7.477, E3 +286542.996}
SPL {X  -159.990, Y  +396.158, Z    +0.000, E1   -12.775, E3 +286543.621}
SPL {X  -159.990, Y  +401.377, Z    +0.000, E1   -19.398, E3 +286544.802}
SPL {X  -159.990, Y  +411.365, Z    +0.000, E1   -30.630, E3 +286548.010}
SPL {X  -159.990, Y  +450.467, Z    +0.000, E1   -50.183, E3 +286571.659}
SPL {X  -159.990, Y  +509.934, Z    +0.000, E1   -54.923, E3 +286634.278}
SPL {X  -159.990, Y  +516.848, Z    +0.000, E1   -54.930, E3 +286644.566}
SPL {X  -159.990, Y  +524.818, Z    +0.000, E1   -54.933, E3 +286656.438}
SPL {X  -159.990, Y  +532.100, Z    +0.000, E1   -54.924, E3 +286667.291}
SPL {X  -159.990, Y  +539.391, Z    +0.000, E1   -54.933, E3 +286678.143}
SPL {X  -159.990, Y  +546.283, Z    +0.000, E1   -54.924, E3 +286688.414}
SPL {X  -159.990, Y  +553.734, Z    +0.000, E1   -54.938, E3 +286699.501}
SPL {X  -159.990, Y  +560.983, Z    +0.000, E1   -54.918, E3 +286710.338}
SPL {X  -159.990, Y  +567.462, Z    +0.000, E1   -54.929, E3 +286719.973}
SPL {X  -159.990, Y  +575.140, Z    +0.000, E1   -54.928, E3 +286731.406}
SPL {X  -159.990, Y  +581.046, Z    +0.000, E1   -54.920, E3 +286740.218}
SPL {X  -159.990, Y  +588.063, Z    +0.000, E1   -54.931, E3 +286750.653}
SPL {X  -159.990, Y  +595.273, Z    +0.000, E1   -54.928, E3 +286761.377}
SPL {X  -159.990, Y  +602.326, Z    +0.000, E1   -54.932, E3 +286771.877}
SPL {X  -159.990, Y  +610.296, Z    +0.000, E1   -54.937, E3 +286783.746}
SPL {X  -159.990, Y  +618.534, Z    +0.000, E1   -54.942, E3 +286795.983}
SPL {X  -159.990, Y  +625.928, Z    +0.000, E1   -54.931, E3 +286807.008}
SPL {X  -159.990, Y  +633.423, Z    +0.000, E1   -54.943, E3 +286818.151}
SPL {X  -159.990, Y  +643.352, Z    +0.000, E1   -54.966, E3 +286832.886}
SPL {X  -159.990, Y  +650.756, Z    +0.000, E1   -54.931, E3 +286843.953}
SPL {X  -159.990, Y  +658.525, Z    +0.000, E1   -54.959, E3 +286855.489}
SPL {X  -159.990, Y  +667.903, Z    +0.000, E1   -54.941, E3 +286869.520}
SPL {X  -159.953, Y  +674.920, Z    +0.000, E1   -54.918, E3 +286880.023}
SPL {X  -159.714, Y  +680.893, Z    +0.000, E1   -54.890, E3 +286889.163}
SPL {X  -159.222, Y  +687.156, Z    +0.000, E1   -54.792, E3 +286899.050}
SPL {X  -158.388, Y  +694.082, Z    +0.000, E1   -54.679, E3 +286910.188}
SPL {X  -157.277, Y  +700.838, Z    +0.000, E1   -54.465, E3 +286921.445}
SPL {X  -156.153, Y  +706.327, Z    +0.000, E1   -54.274, E3 +286930.781}
SPL {X  -154.917, Y  +711.470, Z    +0.000, E1   -54.052, E3 +286939.732}
SPL {X  -153.204, Y  +717.603, Z    +0.000, E1   -53.775, E3 +286950.578}
SPL {X  -151.355, Y  +723.351, Z    +0.000, E1   -53.415, E3 +286961.050}
SPL {X  -149.371, Y  +728.816, Z    +0.000, E1   -53.074, E3 +286971.140}
SPL {X  -146.631, Y  +735.501, Z    +0.000, E1   -52.568, E3 +286983.801}
SPL {X  -144.428, Y  +740.329, Z    +0.000, E1   -52.109, E3 +286993.154}
SPL {X  -142.385, Y  +744.461, Z    +0.000, E1   -51.729, E3 +287001.206}
SPL {X  -132.301, Y  +761.463, Z    +0.000, E1   -45.510, E3 +287078.944}
ENDSPLINE

